LIN {X 0,Y 573.931,Z 295.333,A -85,B 0,C 180,E1 -2262.553,E2 -2262.553} C_VEL
LIN {X 0,Y 573.875,Z 198.299,A -85,B 0,C 180,E1 -2263.776,E2 -2263.776} C_VEL
LIN {X 0,Y 573.396,Z 194.795,A -85,B 0,C 180,E1 -2263.85,E2 -2263.85} C_VEL
LIN {X 0,Y 573.536,Z 174.901,A -85,B 0,C 180,E1 -2266.722,E2 -2266.722} C_VEL
LIN {X 0,Y 573.71,Z 157.017,A -85,B 0,C 180,E1 -2269.314,E2 -2269.314} C_VEL
LIN {X 0,Y 573.882,Z 139.078,A -85,B 0,C 180,E1 -2271.932,E2 -2271.932} C_VEL
LIN {X 0,Y 573.502,Z 133.913,A -85,B 0,C 180,E1 -2272.706,E2 -2272.706} C_VEL
LIN {X 0,Y 573.198,Z 132.088,A -85,B 0,C 180,E1 -2273.017,E2 -2273.017} C_VEL
LIN {X 0,Y 573.2,Z 132.089,A -85,B 0,C 180,E1 -2275.412,E2 -2275.412} C_VEL
LIN {X 0,Y 573.191,Z 132.083,A -85,B 0,C 180,E1 -2278.017,E2 -2278.017} C_VEL
LIN {X 0,Y 573.199,Z 132.085,A -85,B 0,C 180,E1 -2280.877,E2 -2280.877} C_VEL
LIN {X 0,Y 573.24,Z 132.08,A -85,B 0,C 180,E1 -2283.52,E2 -2283.52} C_VEL
LIN {X 0,Y 573.175,Z 132.083,A -85,B 0,C 180,E1 -2286.054,E2 -2286.054} C_VEL
LIN {X 0,Y 573.223,Z 132.081,A -85,B 0,C 180,E1 -2288.702,E2 -2288.702} C_VEL
LIN {X 0,Y 573.19,Z 132.083,A -85,B 0,C 180,E1 -2291.588,E2 -2291.588} C_VEL
LIN {X 0,Y 573.203,Z 132.085,A -85,B 0,C 180,E1 -2294.672,E2 -2294.672} C_VEL
LIN {X 0,Y 573.2,Z 132.08,A -85,B 0,C 180,E1 -2297.596,E2 -2297.596} C_VEL
LIN {X 0,Y 573.225,Z 132.082,A -85,B 0,C 180,E1 -2300.569,E2 -2300.569} C_VEL
LIN {X 0,Y 573.221,Z 132.081,A -85,B 0,C 180,E1 -2303.075,E2 -2303.075} C_VEL
LIN {X 0,Y 573.235,Z 132.075,A -85,B 0,C 180,E1 -2305.669,E2 -2305.669} C_VEL
LIN {X 0,Y 573.212,Z 132.08,A -85,B 0,C 180,E1 -2308.182,E2 -2308.182} C_VEL
LIN {X 0,Y 573.207,Z 132.087,A -85,B 0,C 180,E1 -2310.631,E2 -2310.631} C_VEL
LIN {X 0,Y 573.194,Z 132.079,A -85,B 0,C 180,E1 -2313.514,E2 -2313.514} C_VEL
LIN {X 0,Y 573.184,Z 132.086,A -85,B 0,C 180,E1 -2316.132,E2 -2316.132} C_VEL
LIN {X 0,Y 573.21,Z 132.079,A -85,B 0,C 180,E1 -2319.172,E2 -2319.172} C_VEL
LIN {X 0,Y 573.182,Z 132.081,A -85,B 0,C 180,E1 -2321.41,E2 -2321.41} C_VEL
LIN {X 0,Y 573.194,Z 132.088,A -85,B 0,C 180,E1 -2324.351,E2 -2324.351} C_VEL
LIN {X 0,Y 573.184,Z 132.087,A -85,B 0,C 180,E1 -2326.528,E2 -2326.528} C_VEL
LIN {X 0,Y 573.233,Z 132.075,A -85,B 0,C 180,E1 -2329.402,E2 -2329.402} C_VEL
LIN {X 0,Y 573.21,Z 132.086,A -85,B 0,C 180,E1 -2332.249,E2 -2332.249} C_VEL
LIN {X 0,Y 573.264,Z 132.07,A -85,B 0,C 180,E1 -2335.077,E2 -2335.077} C_VEL
LIN {X 0,Y 573.303,Z 132.075,A -85,B 0,C 180,E1 -2337.892,E2 -2337.892} C_VEL
LIN {X 0,Y 573.309,Z 132.075,A -85,B 0,C 180,E1 -2340,E2 -2340} C_VEL
LIN {X 0,Y 573.261,Z 132.072,A -85,B 0,C 180,E1 -2342.811,E2 -2342.811} C_VEL
LIN {X 0,Y 573.261,Z 132.079,A -85,B 0,C 180,E1 -2345.628,E2 -2345.628} C_VEL
LIN {X 0,Y 573.225,Z 132.078,A -85,B 0,C 180,E1 -2348.46,E2 -2348.46} C_VEL
LIN {X 0,Y 573.226,Z 132.081,A -85,B 0,C 180,E1 -2351.313,E2 -2351.313} C_VEL
LIN {X 0,Y 573.247,Z 132.075,A -85,B 0,C 180,E1 -2354.414,E2 -2354.414} C_VEL
LIN {X 0,Y 573.165,Z 132.088,A -85,B 0,C 180,E1 -2357.114,E2 -2357.114} C_VEL
LIN {X 0,Y 573.255,Z 132.08,A -85,B 0,C 180,E1 -2359.33,E2 -2359.33} C_VEL
LIN {X 0,Y 573.187,Z 132.083,A -85,B 0,C 180,E1 -2362.339,E2 -2362.339} C_VEL
LIN {X 0,Y 573.192,Z 132.086,A -85,B 0,C 180,E1 -2363.279,E2 -2363.279} C_VEL
LIN {X 0,Y 572.863,Z 132.396,A -85,B 0,C 180,E1 -2363.667,E2 -2363.667} C_VEL
LIN {X 0,Y 571.545,Z 133.798,A -85,B 0,C 180,E1 -2364.226,E2 -2364.226} C_VEL
LIN {X 0,Y 569.755,Z 135.989,A -85,B 0,C 180,E1 -2364.752,E2 -2364.752} C_VEL
LIN {X 0,Y 567.024,Z 140.741,A -85,B 0,C 180,E1 -2365.613,E2 -2365.613} C_VEL
LIN {X 0,Y 566.439,Z 143.796,A -85,B 0,C 180,E1 -2366.138,E2 -2366.138} C_VEL
LIN {X 0,Y 566.337,Z 160.929,A -85,B 0,C 180,E1 -2369.129,E2 -2369.129} C_VEL
LIN {X 0,Y 566.28,Z 166.18,A -85,B 0,C 180,E1 -2370.051,E2 -2370.051} C_VEL
LIN {X 0,Y 567.205,Z 173.364,A -85,B 0,C 180,E1 -2370.168,E2 -2370.168} C_VEL
LIN {X 0,Y 566.947,Z 273.932,A -85,B 0,C 180,E1 -2371.466,E2 -2371.466} C_VEL
LIN {X 0,Y 566.823,Z 285.922,A -85,B 0,C 180,E1 -2371.76,E2 -2371.76} C_VEL
LIN {X 0,Y 566.764,Z 296.329,A -85,B 0,C 180,E1 -2372.117,E2 -2372.117} C_VEL
LIN {X 0,Y 566.623,Z 306.781,A -85,B 0,C 180,E1 -2372.583,E2 -2372.583} C_VEL
LIN {X 0,Y 566.446,Z 317.622,A -85,B 0,C 180,E1 -2373.193,E2 -2373.193} C_VEL
LIN {X 0,Y 566.316,Z 329.517,A -85,B 0,C 180,E1 -2374.056,E2 -2374.056} C_VEL
LIN {X 0,Y 566.245,Z 338.018,A -85,B 0,C 180,E1 -2374.815,E2 -2374.815} C_VEL
LIN {X 0,Y 566.139,Z 344.619,A -85,B 0,C 180,E1 -2375.504,E2 -2375.504} C_VEL
LIN {X 0,Y 566.063,Z 351.559,A -85,B 0,C 180,E1 -2376.362,E2 -2376.362} C_VEL
LIN {X 0,Y 565.983,Z 358.32,A -85,B 0,C 180,E1 -2377.374,E2 -2377.374} C_VEL
LIN {X 0,Y 565.975,Z 363.801,A -85,B 0,C 180,E1 -2378.38,E2 -2378.38} C_VEL
LIN {X 0,Y 565.888,Z 367.871,A -85,B 0,C 180,E1 -2379.3,E2 -2379.3} C_VEL
LIN {X 0,Y 565.901,Z 372.701,A -85,B 0,C 180,E1 -2380.751,E2 -2380.751} C_VEL
LIN {X 0,Y 565.861,Z 375.529,A -85,B 0,C 180,E1 -2382.119,E2 -2382.119} C_VEL
LIN {X 0,Y 565.845,Z 376.629,A -85,B 0,C 180,E1 -2383.087,E2 -2383.087} C_VEL
LIN {X 0,Y 565.858,Z 376.999,A -85,B 0,C 180,E1 -2384.069,E2 -2384.069} C_VEL
LIN {X 0,Y 565.875,Z 376.587,A -85,B 0,C 180,E1 -2385.066,E2 -2385.066} C_VEL
LIN {X 0,Y 565.852,Z 375.359,A -85,B 0,C 180,E1 -2386.085,E2 -2386.085} C_VEL
LIN {X 0,Y 565.901,Z 372.206,A -85,B 0,C 180,E1 -2387.505,E2 -2387.505} C_VEL
LIN {X 0,Y 565.921,Z 368.981,A -85,B 0,C 180,E1 -2388.505,E2 -2388.505} C_VEL
LIN {X 0,Y 565.944,Z 364.768,A -85,B 0,C 180,E1 -2389.512,E2 -2389.512} C_VEL
LIN {X 0,Y 566.014,Z 359.438,A -85,B 0,C 180,E1 -2390.528,E2 -2390.528} C_VEL
LIN {X 0,Y 566.022,Z 353.429,A -85,B 0,C 180,E1 -2391.465,E2 -2391.465} C_VEL
LIN {X 0,Y 566.111,Z 346.956,A -85,B 0,C 180,E1 -2392.309,E2 -2392.309} C_VEL
LIN {X 0,Y 566.208,Z 339.781,A -85,B 0,C 180,E1 -2393.099,E2 -2393.099} C_VEL
LIN {X 0,Y 566.346,Z 332.677,A -85,B 0,C 180,E1 -2393.765,E2 -2393.765} C_VEL
LIN {X 0,Y 566.39,Z 324.604,A -85,B 0,C 180,E1 -2394.413,E2 -2394.413} C_VEL
LIN {X 0,Y 566.516,Z 315.348,A -85,B 0,C 180,E1 -2395.031,E2 -2395.031} C_VEL
LIN {X 0,Y 566.609,Z 306.216,A -85,B 0,C 180,E1 -2395.535,E2 -2395.535} C_VEL
LIN {X 0,Y 566.726,Z 296.359,A -85,B 0,C 180,E1 -2395.973,E2 -2395.973} C_VEL
LIN {X 0,Y 566.82,Z 285.576,A -85,B 0,C 180,E1 -2396.34,E2 -2396.34} C_VEL
LIN {X 0,Y 566.935,Z 273.792,A -85,B 0,C 180,E1 -2396.627,E2 -2396.627} C_VEL
LIN {X 0,Y 567.061,Z 171.116,A -85,B 0,C 180,E1 -2397.954,E2 -2397.954} C_VEL
LIN {X 0,Y 566.232,Z 166.076,A -85,B 0,C 180,E1 -2398.059,E2 -2398.059} C_VEL
LIN {X 0,Y 566.436,Z 150.118,A -85,B 0,C 180,E1 -2400.87,E2 -2400.87} C_VEL
LIN {X 0,Y 566.555,Z 135.482,A -85,B 0,C 180,E1 -2403.477,E2 -2403.477} C_VEL
LIN {X 0,Y 566.18,Z 132.961,A -85,B 0,C 180,E1 -2403.953,E2 -2403.953} C_VEL
LIN {X 0,Y 566.142,Z 132.968,A -85,B 0,C 180,E1 -2406.725,E2 -2406.725} C_VEL
LIN {X 0,Y 566.184,Z 132.958,A -85,B 0,C 180,E1 -2408.902,E2 -2408.902} C_VEL
LIN {X 0,Y 566.177,Z 132.955,A -85,B 0,C 180,E1 -2411.172,E2 -2411.172} C_VEL
LIN {X 0,Y 566.164,Z 132.961,A -85,B 0,C 180,E1 -2414.152,E2 -2414.152} C_VEL
LIN {X 0,Y 566.156,Z 132.966,A -85,B 0,C 180,E1 -2416.358,E2 -2416.358} C_VEL
LIN {X 0,Y 566.206,Z 132.95,A -85,B 0,C 180,E1 -2419.27,E2 -2419.27} C_VEL
LIN {X 0,Y 566.183,Z 132.961,A -85,B 0,C 180,E1 -2422.152,E2 -2422.152} C_VEL
LIN {X 0,Y 566.245,Z 132.946,A -85,B 0,C 180,E1 -2425.016,E2 -2425.016} C_VEL
LIN {X 0,Y 566.275,Z 132.947,A -85,B 0,C 180,E1 -2427.866,E2 -2427.866} C_VEL
LIN {X 0,Y 566.282,Z 132.949,A -85,B 0,C 180,E1 -2430,E2 -2430} C_VEL
LIN {X 0,Y 566.234,Z 132.947,A -85,B 0,C 180,E1 -2432.846,E2 -2432.846} C_VEL
LIN {X 0,Y 566.232,Z 132.953,A -85,B 0,C 180,E1 -2435.699,E2 -2435.699} C_VEL
LIN {X 0,Y 566.182,Z 132.954,A -85,B 0,C 180,E1 -2438.566,E2 -2438.566} C_VEL
LIN {X 0,Y 566.189,Z 132.956,A -85,B 0,C 180,E1 -2441.455,E2 -2441.455} C_VEL
LIN {X 0,Y 566.199,Z 132.952,A -85,B 0,C 180,E1 -2444.494,E2 -2444.494} C_VEL
LIN {X 0,Y 566.153,Z 132.961,A -85,B 0,C 180,E1 -2447.333,E2 -2447.333} C_VEL
LIN {X 0,Y 566.17,Z 132.964,A -85,B 0,C 180,E1 -2449.582,E2 -2449.582} C_VEL
LIN {X 0,Y 566.141,Z 132.964,A -85,B 0,C 180,E1 -2451.864,E2 -2451.864} C_VEL
LIN {X 0,Y 566.174,Z 132.957,A -85,B 0,C 180,E1 -2455.021,E2 -2455.021} C_VEL
LIN {X 0,Y 566.154,Z 132.965,A -85,B 0,C 180,E1 -2457.342,E2 -2457.342} C_VEL
LIN {X 0,Y 566.142,Z 132.963,A -85,B 0,C 180,E1 -2459.772,E2 -2459.772} C_VEL
LIN {X 0,Y 566.185,Z 132.953,A -85,B 0,C 180,E1 -2462.427,E2 -2462.427} C_VEL
LIN {X 0,Y 566.156,Z 132.961,A -85,B 0,C 180,E1 -2464.986,E2 -2464.986} C_VEL
LIN {X 0,Y 566.182,Z 132.96,A -85,B 0,C 180,E1 -2467.461,E2 -2467.461} C_VEL
LIN {X 0,Y 566.188,Z 132.953,A -85,B 0,C 180,E1 -2470.2,E2 -2470.2} C_VEL
LIN {X 0,Y 566.17,Z 132.964,A -85,B 0,C 180,E1 -2473.056,E2 -2473.056} C_VEL
LIN {X 0,Y 566.148,Z 132.957,A -85,B 0,C 180,E1 -2476.053,E2 -2476.053} C_VEL
LIN {X 0,Y 566.148,Z 132.965,A -85,B 0,C 180,E1 -2478.858,E2 -2478.858} C_VEL
LIN {X 0,Y 566.191,Z 132.955,A -85,B 0,C 180,E1 -2481.444,E2 -2481.444} C_VEL
LIN {X 0,Y 566.128,Z 132.962,A -85,B 0,C 180,E1 -2484.306,E2 -2484.306} C_VEL
LIN {X 0,Y 566.184,Z 132.962,A -85,B 0,C 180,E1 -2486.896,E2 -2486.896} C_VEL
LIN {X 0,Y 566.15,Z 132.959,A -85,B 0,C 180,E1 -2489.406,E2 -2489.406} C_VEL
LIN {X 0,Y 566.133,Z 132.96,A -85,B 0,C 180,E1 -2491.854,E2 -2491.854} C_VEL
LIN {X 0,Y 566.179,Z 132.957,A -85,B 0,C 180,E1 -2494.25,E2 -2494.25} C_VEL
LIN {X 0,Y 566.13,Z 132.96,A -85,B 0,C 180,E1 -2497.367,E2 -2497.367} C_VEL
LIN {X 0,Y 566.16,Z 132.956,A -85,B 0,C 180,E1 -2499.661,E2 -2499.661} C_VEL
LIN {X 0,Y 566.153,Z 132.959,A -85,B 0,C 180,E1 -2501.921,E2 -2501.921} C_VEL
LIN {X 0,Y 566.171,Z 132.957,A -85,B 0,C 180,E1 -2504.89,E2 -2504.89} C_VEL
LIN {X 0,Y 566.164,Z 132.958,A -85,B 0,C 180,E1 -2507.818,E2 -2507.818} C_VEL
LIN {X 0,Y 566.152,Z 132.962,A -85,B 0,C 180,E1 -2509.992,E2 -2509.992} C_VEL
LIN {X 0,Y 566.175,Z 132.955,A -85,B 0,C 180,E1 -2512.87,E2 -2512.87} C_VEL
LIN {X 0,Y 566.242,Z 132.946,A -85,B 0,C 180,E1 -2515.016,E2 -2515.016} C_VEL
LIN {X 0,Y 566.273,Z 132.948,A -85,B 0,C 180,E1 -2517.867,E2 -2517.867} C_VEL
LIN {X 0,Y 566.279,Z 132.95,A -85,B 0,C 180,E1 -2520,E2 -2520} C_VEL
LIN {X 0,Y 566.231,Z 132.947,A -85,B 0,C 180,E1 -2522.846,E2 -2522.846} C_VEL
LIN {X 0,Y 566.23,Z 132.953,A -85,B 0,C 180,E1 -2525.699,E2 -2525.699} C_VEL
LIN {X 0,Y 566.179,Z 132.955,A -85,B 0,C 180,E1 -2528.567,E2 -2528.567} C_VEL
LIN {X 0,Y 566.186,Z 132.957,A -85,B 0,C 180,E1 -2531.456,E2 -2531.456} C_VEL
LIN {X 0,Y 566.197,Z 132.952,A -85,B 0,C 180,E1 -2534.494,E2 -2534.494} C_VEL
LIN {X 0,Y 566.151,Z 132.962,A -85,B 0,C 180,E1 -2537.333,E2 -2537.333} C_VEL
LIN {X 0,Y 566.168,Z 132.965,A -85,B 0,C 180,E1 -2539.582,E2 -2539.582} C_VEL
LIN {X 0,Y 566.14,Z 132.964,A -85,B 0,C 180,E1 -2541.865,E2 -2541.865} C_VEL
LIN {X 0,Y 566.173,Z 132.957,A -85,B 0,C 180,E1 -2545.022,E2 -2545.022} C_VEL
LIN {X 0,Y 566.153,Z 132.965,A -85,B 0,C 180,E1 -2547.342,E2 -2547.342} C_VEL
LIN {X 0,Y 566.141,Z 132.962,A -85,B 0,C 180,E1 -2549.773,E2 -2549.773} C_VEL
LIN {X 0,Y 566.185,Z 132.953,A -85,B 0,C 180,E1 -2552.428,E2 -2552.428} C_VEL
LIN {X 0,Y 566.154,Z 132.962,A -85,B 0,C 180,E1 -2554.987,E2 -2554.987} C_VEL
LIN {X 0,Y 566.184,Z 132.959,A -85,B 0,C 180,E1 -2557.462,E2 -2557.462} C_VEL
LIN {X 0,Y 566.162,Z 132.956,A -85,B 0,C 180,E1 -2560.203,E2 -2560.203} C_VEL
LIN {X 0,Y 566.144,Z 132.968,A -85,B 0,C 180,E1 -2563.06,E2 -2563.06} C_VEL
LIN {X 0,Y 566.151,Z 132.957,A -85,B 0,C 180,E1 -2566.054,E2 -2566.054} C_VEL
LIN {X 0,Y 566.141,Z 132.967,A -85,B 0,C 180,E1 -2568.858,E2 -2568.858} C_VEL
LIN {X 0,Y 566.168,Z 132.956,A -85,B 0,C 180,E1 -2571.636,E2 -2571.636} C_VEL
LIN {X 0,Y 566.129,Z 132.962,A -85,B 0,C 180,E1 -2574.306,E2 -2574.306} C_VEL
LIN {X 0,Y 566.16,Z 132.965,A -85,B 0,C 180,E1 -2576.894,E2 -2576.894} C_VEL
LIN {X 0,Y 566.147,Z 132.959,A -85,B 0,C 180,E1 -2579.406,E2 -2579.406} C_VEL
LIN {X 0,Y 566.139,Z 132.96,A -85,B 0,C 180,E1 -2581.854,E2 -2581.854} C_VEL
LIN {X 0,Y 566.171,Z 132.959,A -85,B 0,C 180,E1 -2584.249,E2 -2584.249} C_VEL
LIN {X 0,Y 566.158,Z 133.045,A -85,B 0,C 180,E1 -2586.833,E2 -2586.833} C_VEL
LIN {X 0,Y 566.938,Z 137.862,A -85,B 0,C 180,E1 -2587.593,E2 -2587.593} C_VEL
LIN {X 0,Y 566.777,Z 155.67,A -85,B 0,C 180,E1 -2590.251,E2 -2590.251} C_VEL
LIN {X 0,Y 566.546,Z 172.886,A -85,B 0,C 180,E1 -2592.783,E2 -2592.783} C_VEL
LIN {X 0,Y 566.406,Z 192.432,A -85,B 0,C 180,E1 -2595.631,E2 -2595.631} C_VEL
LIN {X 0,Y 566.422,Z 195.149,A -85,B 0,C 180,E1 -2595.998,E2 -2595.998} C_VEL
LIN {X 0,Y 567.176,Z 200.341,A -85,B 0,C 180,E1 -2596.084,E2 -2596.084} C_VEL
LIN {X 0,Y 566.98,Z 302.95,A -85,B 0,C 180,E1 -2597.404,E2 -2597.404} C_VEL
LIN {X 0,Y 566.841,Z 316.219,A -85,B 0,C 180,E1 -2597.719,E2 -2597.719} C_VEL
LIN {X 0,Y 566.743,Z 328.379,A -85,B 0,C 180,E1 -2598.148,E2 -2598.148} C_VEL
LIN {X 0,Y 566.603,Z 340.366,A -85,B 0,C 180,E1 -2598.72,E2 -2598.72} C_VEL
LIN {X 0,Y 566.439,Z 352.196,A -85,B 0,C 180,E1 -2599.455,E2 -2599.455} C_VEL
LIN {X 0,Y 566.325,Z 362.605,A -85,B 0,C 180,E1 -2600.265,E2 -2600.265} C_VEL
LIN {X 0,Y 566.207,Z 371.113,A -85,B 0,C 180,E1 -2601.074,E2 -2601.074} C_VEL
LIN {X 0,Y 566.112,Z 378.961,A -85,B 0,C 180,E1 -2601.972,E2 -2601.972} C_VEL
LIN {X 0,Y 566.004,Z 386.623,A -85,B 0,C 180,E1 -2603.047,E2 -2603.047} C_VEL
LIN {X 0,Y 566.004,Z 393.679,A -85,B 0,C 180,E1 -2604.299,E2 -2604.299} C_VEL
LIN {X 0,Y 565.933,Z 398.372,A -85,B 0,C 180,E1 -2605.37,E2 -2605.37} C_VEL
LIN {X 0,Y 565.927,Z 401.958,A -85,B 0,C 180,E1 -2606.44,E2 -2606.44} C_VEL
LIN {X 0,Y 565.878,Z 403.807,A -85,B 0,C 180,E1 -2607.152,E2 -2607.152} C_VEL
LIN {X 0,Y 565.846,Z 406.184,A -85,B 0,C 180,E1 -2608.576,E2 -2608.576} C_VEL
LIN {X 0,Y 565.839,Z 407,A -85,B 0,C 180,E1 -2610,E2 -2610} C_VEL
LIN {X 0,Y 565.846,Z 406.185,A -85,B 0,C 180,E1 -2611.423,E2 -2611.423} C_VEL
LIN {X 0,Y 565.878,Z 403.81,A -85,B 0,C 180,E1 -2612.847,E2 -2612.847} C_VEL
LIN {X 0,Y 565.926,Z 400.896,A -85,B 0,C 180,E1 -2613.916,E2 -2613.916} C_VEL
LIN {X 0,Y 565.878,Z 396.949,A -85,B 0,C 180,E1 -2614.987,E2 -2614.987} C_VEL
LIN {X 0,Y 566.002,Z 391.868,A -85,B 0,C 180,E1 -2616.058,E2 -2616.058} C_VEL
LIN {X 0,Y 566.04,Z 385.469,A -85,B 0,C 180,E1 -2617.132,E2 -2617.132} C_VEL
LIN {X 0,Y 566.134,Z 377.479,A -85,B 0,C 180,E1 -2618.207,E2 -2618.207} C_VEL
LIN {X 0,Y 566.229,Z 369.336,A -85,B 0,C 180,E1 -2619.105,E2 -2619.105} C_VEL
LIN {X 0,Y 566.347,Z 359.402,A -85,B 0,C 180,E1 -2620.005,E2 -2620.005} C_VEL
LIN {X 0,Y 566.536,Z 348.295,A -85,B 0,C 180,E1 -2620.807,E2 -2620.807} C_VEL
LIN {X 0,Y 566.612,Z 337.178,A -85,B 0,C 180,E1 -2621.446,E2 -2621.446} C_VEL
LIN {X 0,Y 566.745,Z 324.986,A -85,B 0,C 180,E1 -2621.988,E2 -2621.988} C_VEL
LIN {X 0,Y 566.917,Z 312.186,A -85,B 0,C 180,E1 -2622.393,E2 -2622.393} C_VEL
LIN {X 0,Y 566.994,Z 300.124,A -85,B 0,C 180,E1 -2622.641,E2 -2622.641} C_VEL
LIN {X 0,Y 567.04,Z 199.447,A -85,B 0,C 180,E1 -2623.931,E2 -2623.931} C_VEL
LIN {X 0,Y 566.391,Z 194.795,A -85,B 0,C 180,E1 -2624.025,E2 -2624.025} C_VEL
LIN {X 0,Y 566.55,Z 175.031,A -85,B 0,C 180,E1 -2626.895,E2 -2626.895} C_VEL
LIN {X 0,Y 566.73,Z 156.765,A -85,B 0,C 180,E1 -2629.562,E2 -2629.562} C_VEL
LIN {X 0,Y 566.912,Z 138.815,A -85,B 0,C 180,E1 -2632.216,E2 -2632.216} C_VEL
LIN {X 0,Y 566.155,Z 132.966,A -85,B 0,C 180,E1 -2633.142,E2 -2633.142} C_VEL
LIN {X 0,Y 566.17,Z 132.961,A -85,B 0,C 180,E1 -2635.751,E2 -2635.751} C_VEL
LIN {X 0,Y 566.136,Z 132.961,A -85,B 0,C 180,E1 -2638.189,E2 -2638.189} C_VEL
LIN {X 0,Y 566.167,Z 132.964,A -85,B 0,C 180,E1 -2641.072,E2 -2641.072} C_VEL
LIN {X 0,Y 566.193,Z 132.955,A -85,B 0,C 180,E1 -2643.731,E2 -2643.731} C_VEL
LIN {X 0,Y 566.142,Z 132.961,A -85,B 0,C 180,E1 -2646.573,E2 -2646.573} C_VEL
LIN {X 0,Y 566.199,Z 132.959,A -85,B 0,C 180,E1 -2649.274,E2 -2649.274} C_VEL
LIN {X 0,Y 566.139,Z 132.96,A -85,B 0,C 180,E1 -2652.093,E2 -2652.093} C_VEL
LIN {X 0,Y 566.16,Z 132.965,A -85,B 0,C 180,E1 -2655.036,E2 -2655.036} C_VEL
LIN {X 0,Y 566.136,Z 132.96,A -85,B 0,C 180,E1 -2658.144,E2 -2658.144} C_VEL
LIN {X 0,Y 566.197,Z 132.96,A -85,B 0,C 180,E1 -2660.725,E2 -2660.725} C_VEL
LIN {X 0,Y 566.142,Z 132.959,A -85,B 0,C 180,E1 -2663.425,E2 -2663.425} C_VEL
LIN {X 0,Y 566.189,Z 132.956,A -85,B 0,C 180,E1 -2666.268,E2 -2666.268} C_VEL
LIN {X 0,Y 566.165,Z 132.96,A -85,B 0,C 180,E1 -2668.926,E2 -2668.926} C_VEL
LIN {X 0,Y 566.133,Z 132.96,A -85,B 0,C 180,E1 -2671.853,E2 -2671.853} C_VEL
LIN {X 0,Y 566.18,Z 132.958,A -85,B 0,C 180,E1 -2674.249,E2 -2674.249} C_VEL
LIN {X 0,Y 566.14,Z 132.963,A -85,B 0,C 180,E1 -2676.724,E2 -2676.724} C_VEL
LIN {X 0,Y 566.175,Z 132.957,A -85,B 0,C 180,E1 -2678.901,E2 -2678.901} C_VEL
LIN {X 0,Y 566.159,Z 132.956,A -85,B 0,C 180,E1 -2681.17,E2 -2681.17} C_VEL
LIN {X 0,Y 566.161,Z 132.964,A -85,B 0,C 180,E1 -2684.151,E2 -2684.151} C_VEL
LIN {X 0,Y 566.152,Z 132.966,A -85,B 0,C 180,E1 -2686.357,E2 -2686.357} C_VEL
LIN {X 0,Y 566.203,Z 132.951,A -85,B 0,C 180,E1 -2689.269,E2 -2689.269} C_VEL
LIN {X 0,Y 566.178,Z 132.963,A -85,B 0,C 180,E1 -2692.152,E2 -2692.152} C_VEL
LIN {X 0,Y 566.24,Z 132.945,A -85,B 0,C 180,E1 -2695.015,E2 -2695.015} C_VEL
LIN {X 0,Y 566.272,Z 132.95,A -85,B 0,C 180,E1 -2697.866,E2 -2697.866} C_VEL
LIN {X 0,Y 566.277,Z 132.95,A -85,B 0,C 180,E1 -2700,E2 -2700} C_VEL
LIN {X 0,Y 566.229,Z 132.948,A -85,B 0,C 180,E1 -2702.845,E2 -2702.845} C_VEL
LIN {X 0,Y 566.23,Z 132.956,A -85,B 0,C 180,E1 -2705.698,E2 -2705.698} C_VEL
LIN {X 0,Y 566.177,Z 132.955,A -85,B 0,C 180,E1 -2708.566,E2 -2708.566} C_VEL
LIN {X 0,Y 566.183,Z 132.961,A -85,B 0,C 180,E1 -2711.455,E2 -2711.455} C_VEL
LIN {X 0,Y 566.203,Z 132.953,A -85,B 0,C 180,E1 -2714.497,E2 -2714.497} C_VEL
LIN {X 0,Y 566.139,Z 132.966,A -85,B 0,C 180,E1 -2717.333,E2 -2717.333} C_VEL
LIN {X 0,Y 566.187,Z 132.963,A -85,B 0,C 180,E1 -2719.581,E2 -2719.581} C_VEL
LIN {X 0,Y 566.14,Z 132.965,A -85,B 0,C 180,E1 -2721.864,E2 -2721.864} C_VEL
LIN {X 0,Y 566.179,Z 133.046,A -85,B 0,C 180,E1 -2724.279,E2 -2724.279} C_VEL
LIN {X 0,Y 566.495,Z 137.739,A -85,B 0,C 180,E1 -2725.092,E2 -2725.092} C_VEL
LIN {X 0,Y 566.439,Z 143.796,A -85,B 0,C 180,E1 -2726.138,E2 -2726.138} C_VEL
LIN {X 0,Y 565.819,Z 146.819,A -85,B 0,C 180,E1 -2726.647,E2 -2726.647} C_VEL
LIN {X 0,Y 562.955,Z 151.99,A -85,B 0,C 180,E1 -2727.456,E2 -2727.456} C_VEL
LIN {X 0,Y 560.027,Z 157.182,A -85,B 0,C 180,E1 -2728.272,E2 -2728.272} C_VEL
LIN {X 0,Y 559.328,Z 160.192,A -85,B 0,C 180,E1 -2728.789,E2 -2728.789} C_VEL
LIN {X 0,Y 559.233,Z 166.292,A -85,B 0,C 180,E1 -2729.874,E2 -2729.874} C_VEL
LIN {X 0,Y 560.329,Z 174.113,A -85,B 0,C 180,E1 -2730.004,E2 -2730.004} C_VEL
LIN {X 0,Y 560.055,Z 273.245,A -85,B 0,C 180,E1 -2731.296,E2 -2731.296} C_VEL
LIN {X 0,Y 559.909,Z 284.947,A -85,B 0,C 180,E1 -2731.578,E2 -2731.578} C_VEL
LIN {X 0,Y 559.807,Z 295.31,A -85,B 0,C 180,E1 -2731.927,E2 -2731.927} C_VEL
LIN {X 0,Y 559.67,Z 305.191,A -85,B 0,C 180,E1 -2732.361,E2 -2732.361} C_VEL
LIN {X 0,Y 559.524,Z 314.402,A -85,B 0,C 180,E1 -2732.864,E2 -2732.864} C_VEL
LIN {X 0,Y 559.4,Z 323.117,A -85,B 0,C 180,E1 -2733.44,E2 -2733.44} C_VEL
LIN {X 0,Y 559.308,Z 330.635,A -85,B 0,C 180,E1 -2734.026,E2 -2734.026} C_VEL
LIN {X 0,Y 559.195,Z 338.709,A -85,B 0,C 180,E1 -2734.769,E2 -2734.769} C_VEL
LIN {X 0,Y 559.095,Z 345.863,A -85,B 0,C 180,E1 -2735.547,E2 -2735.547} C_VEL
LIN {X 0,Y 558.995,Z 352.677,A -85,B 0,C 180,E1 -2736.426,E2 -2736.426} C_VEL
LIN {X 0,Y 558.911,Z 358.761,A -85,B 0,C 180,E1 -2737.366,E2 -2737.366} C_VEL
LIN {X 0,Y 558.892,Z 364.246,A -85,B 0,C 180,E1 -2738.403,E2 -2738.403} C_VEL
LIN {X 0,Y 558.802,Z 368.591,A -85,B 0,C 180,E1 -2739.429,E2 -2739.429} C_VEL
LIN {X 0,Y 558.806,Z 371.692,A -85,B 0,C 180,E1 -2740.368,E2 -2740.368} C_VEL
LIN {X 0,Y 558.788,Z 373.433,A -85,B 0,C 180,E1 -2741.008,E2 -2741.008} C_VEL
LIN {X 0,Y 558.761,Z 375.515,A -85,B 0,C 180,E1 -2742.091,E2 -2742.091} C_VEL
LIN {X 0,Y 558.759,Z 376.672,A -85,B 0,C 180,E1 -2743.155,E2 -2743.155} C_VEL
LIN {X 0,Y 558.774,Z 376.972,A -85,B 0,C 180,E1 -2744.2,E2 -2744.2} C_VEL
LIN {X 0,Y 558.784,Z 376.456,A -85,B 0,C 180,E1 -2745.226,E2 -2745.226} C_VEL
LIN {X 0,Y 558.76,Z 375.174,A -85,B 0,C 180,E1 -2746.23,E2 -2746.23} C_VEL
LIN {X 0,Y 558.773,Z 373.114,A -85,B 0,C 180,E1 -2747.221,E2 -2747.221} C_VEL
LIN {X 0,Y 558.823,Z 370.284,A -85,B 0,C 180,E1 -2748.2,E2 -2748.2} C_VEL
LIN {X 0,Y 558.862,Z 365.631,A -85,B 0,C 180,E1 -2749.4,E2 -2749.4} C_VEL
LIN {X 0,Y 558.939,Z 359.588,A -85,B 0,C 180,E1 -2750.583,E2 -2750.583} C_VEL
LIN {X 0,Y 558.971,Z 354.502,A -85,B 0,C 180,E1 -2751.405,E2 -2751.405} C_VEL
LIN {X 0,Y 559.044,Z 347.29,A -85,B 0,C 180,E1 -2752.372,E2 -2752.372} C_VEL
LIN {X 0,Y 559.161,Z 341.184,A -85,B 0,C 180,E1 -2753.07,E2 -2753.07} C_VEL
LIN {X 0,Y 559.305,Z 332.375,A -85,B 0,C 180,E1 -2753.914,E2 -2753.914} C_VEL
LIN {X 0,Y 559.395,Z 324.008,A -85,B 0,C 180,E1 -2754.586,E2 -2754.586} C_VEL
LIN {X 0,Y 559.516,Z 315.753,A -85,B 0,C 180,E1 -2755.145,E2 -2755.145} C_VEL
LIN {X 0,Y 559.638,Z 306.899,A -85,B 0,C 180,E1 -2755.645,E2 -2755.645} C_VEL
LIN {X 0,Y 559.768,Z 296.43,A -85,B 0,C 180,E1 -2756.12,E2 -2756.12} C_VEL
LIN {X 0,Y 559.884,Z 286.241,A -85,B 0,C 180,E1 -2756.475,E2 -2756.475} C_VEL
LIN {X 0,Y 560.016,Z 274.242,A -85,B 0,C 180,E1 -2756.776,E2 -2756.776} C_VEL
LIN {X 0,Y 560.169,Z 217.742,A -85,B 0,C 180,E1 -2757.525,E2 -2757.525} C_VEL
LIN {X 0,Y 560.172,Z 171.726,A -85,B 0,C 180,E1 -2758.123,E2 -2758.123} C_VEL
LIN {X 0,Y 559.232,Z 166.277,A -85,B 0,C 180,E1 -2758.221,E2 -2758.221} C_VEL
LIN {X 0,Y 559.426,Z 150.276,A -85,B 0,C 180,E1 -2761.075,E2 -2761.075} C_VEL
LIN {X 0,Y 559.571,Z 136.646,A -85,B 0,C 180,E1 -2763.522,E2 -2763.522} C_VEL
LIN {X 0,Y 559.147,Z 133.838,A -85,B 0,C 180,E1 -2764.052,E2 -2764.052} C_VEL
LIN {X 0,Y 559.086,Z 133.842,A -85,B 0,C 180,E1 -2767.066,E2 -2767.066} C_VEL
LIN {X 0,Y 559.142,Z 133.831,A -85,B 0,C 180,E1 -2769.394,E2 -2769.394} C_VEL
LIN {X 0,Y 559.108,Z 133.835,A -85,B 0,C 180,E1 -2771.685,E2 -2771.685} C_VEL
LIN {X 0,Y 559.123,Z 133.838,A -85,B 0,C 180,E1 -2774.695,E2 -2774.695} C_VEL
LIN {X 0,Y 559.136,Z 133.832,A -85,B 0,C 180,E1 -2777.662,E2 -2777.662} C_VEL
LIN {X 0,Y 559.114,Z 133.837,A -85,B 0,C 180,E1 -2779.865,E2 -2779.865} C_VEL
LIN {X 0,Y 559.145,Z 133.832,A -85,B 0,C 180,E1 -2782.78,E2 -2782.78} C_VEL
LIN {X 0,Y 559.222,Z 133.821,A -85,B 0,C 180,E1 -2784.953,E2 -2784.953} C_VEL
LIN {X 0,Y 559.245,Z 133.822,A -85,B 0,C 180,E1 -2787.84,E2 -2787.84} C_VEL
LIN {X 0,Y 559.25,Z 133.825,A -85,B 0,C 180,E1 -2790,E2 -2790} C_VEL
LIN {X 0,Y 559.202,Z 133.823,A -85,B 0,C 180,E1 -2792.882,E2 -2792.882} C_VEL
LIN {X 0,Y 559.201,Z 133.83,A -85,B 0,C 180,E1 -2795.77,E2 -2795.77} C_VEL
LIN {X 0,Y 559.147,Z 133.83,A -85,B 0,C 180,E1 -2798.675,E2 -2798.675} C_VEL
LIN {X 0,Y 559.151,Z 133.835,A -85,B 0,C 180,E1 -2801.602,E2 -2801.602} C_VEL
LIN {X 0,Y 559.149,Z 133.83,A -85,B 0,C 180,E1 -2804.576,E2 -2804.576} C_VEL
LIN {X 0,Y 559.108,Z 133.842,A -85,B 0,C 180,E1 -2807.558,E2 -2807.558} C_VEL
LIN {X 0,Y 559.132,Z 133.838,A -85,B 0,C 180,E1 -2809.839,E2 -2809.839} C_VEL
LIN {X 0,Y 559.097,Z 133.838,A -85,B 0,C 180,E1 -2812.154,E2 -2812.154} C_VEL
LIN {X 0,Y 559.134,Z 133.836,A -85,B 0,C 180,E1 -2815.178,E2 -2815.178} C_VEL
LIN {X 0,Y 559.095,Z 133.842,A -85,B 0,C 180,E1 -2817.716,E2 -2817.716} C_VEL
LIN {X 0,Y 559.089,Z 133.837,A -85,B 0,C 180,E1 -2820.186,E2 -2820.186} C_VEL
LIN {X 0,Y 559.141,Z 133.832,A -85,B 0,C 180,E1 -2822.716,E2 -2822.716} C_VEL
LIN {X 0,Y 559.108,Z 133.844,A -85,B 0,C 180,E1 -2825.325,E2 -2825.325} C_VEL
LIN {X 0,Y 559.116,Z 133.834,A -85,B 0,C 180,E1 -2828.018,E2 -2828.018} C_VEL
LIN {X 0,Y 559.143,Z 133.831,A -85,B 0,C 180,E1 -2829.94,E2 -2829.94} C_VEL
LIN {X 0,Y 559.116,Z 133.842,A -85,B 0,C 180,E1 -2833.194,E2 -2833.194} C_VEL
LIN {X 0,Y 559.116,Z 133.834,A -85,B 0,C 180,E1 -2835.764,E2 -2835.764} C_VEL
LIN {X 0,Y 559.093,Z 133.837,A -85,B 0,C 180,E1 -2838.224,E2 -2838.224} C_VEL
LIN {X 0,Y 559.16,Z 133.836,A -85,B 0,C 180,E1 -2841.065,E2 -2841.065} C_VEL
LIN {X 0,Y 559.105,Z 133.835,A -85,B 0,C 180,E1 -2843.787,E2 -2843.787} C_VEL
LIN {X 0,Y 559.136,Z 133.835,A -85,B 0,C 180,E1 -2846.424,E2 -2846.424} C_VEL
LIN {X 0,Y 559.134,Z 133.838,A -85,B 0,C 180,E1 -2848.98,E2 -2848.98} C_VEL
LIN {X 0,Y 559.095,Z 133.836,A -85,B 0,C 180,E1 -2851.632,E2 -2851.632} C_VEL
LIN {X 0,Y 559.145,Z 133.831,A -85,B 0,C 180,E1 -2853.901,E2 -2853.901} C_VEL
LIN {X 0,Y 559.088,Z 133.84,A -85,B 0,C 180,E1 -2857.065,E2 -2857.065} C_VEL
LIN {X 0,Y 559.139,Z 133.831,A -85,B 0,C 180,E1 -2859.394,E2 -2859.394} C_VEL
LIN {X 0,Y 559.105,Z 133.835,A -85,B 0,C 180,E1 -2861.685,E2 -2861.685} C_VEL
LIN {X 0,Y 559.12,Z 133.838,A -85,B 0,C 180,E1 -2864.695,E2 -2864.695} C_VEL
LIN {X 0,Y 559.133,Z 133.833,A -85,B 0,C 180,E1 -2867.662,E2 -2867.662} C_VEL
LIN {X 0,Y 559.111,Z 133.837,A -85,B 0,C 180,E1 -2869.865,E2 -2869.865} C_VEL
LIN {X 0,Y 559.141,Z 133.832,A -85,B 0,C 180,E1 -2872.78,E2 -2872.78} C_VEL
LIN {X 0,Y 559.219,Z 133.821,A -85,B 0,C 180,E1 -2874.953,E2 -2874.953} C_VEL
LIN {X 0,Y 559.243,Z 133.823,A -85,B 0,C 180,E1 -2877.84,E2 -2877.84} C_VEL
LIN {X 0,Y 559.247,Z 133.826,A -85,B 0,C 180,E1 -2880,E2 -2880} C_VEL
LIN {X 0,Y 559.199,Z 133.823,A -85,B 0,C 180,E1 -2882.882,E2 -2882.882} C_VEL
LIN {X 0,Y 559.199,Z 133.83,A -85,B 0,C 180,E1 -2885.771,E2 -2885.771} C_VEL
LIN {X 0,Y 559.144,Z 133.83,A -85,B 0,C 180,E1 -2888.675,E2 -2888.675} C_VEL
LIN {X 0,Y 559.148,Z 133.836,A -85,B 0,C 180,E1 -2891.602,E2 -2891.602} C_VEL
LIN {X 0,Y 559.147,Z 133.83,A -85,B 0,C 180,E1 -2894.577,E2 -2894.577} C_VEL
LIN {X 0,Y 559.106,Z 133.843,A -85,B 0,C 180,E1 -2897.559,E2 -2897.559} C_VEL
LIN {X 0,Y 559.13,Z 133.838,A -85,B 0,C 180,E1 -2899.839,E2 -2899.839} C_VEL
LIN {X 0,Y 559.095,Z 133.838,A -85,B 0,C 180,E1 -2902.155,E2 -2902.155} C_VEL
LIN {X 0,Y 559.134,Z 133.836,A -85,B 0,C 180,E1 -2905.178,E2 -2905.178} C_VEL
LIN {X 0,Y 559.095,Z 133.841,A -85,B 0,C 180,E1 -2907.717,E2 -2907.717} C_VEL
LIN {X 0,Y 559.087,Z 133.837,A -85,B 0,C 180,E1 -2910.187,E2 -2910.187} C_VEL
LIN {X 0,Y 559.142,Z 133.832,A -85,B 0,C 180,E1 -2912.717,E2 -2912.717} C_VEL
LIN {X 0,Y 559.108,Z 133.844,A -85,B 0,C 180,E1 -2915.326,E2 -2915.326} C_VEL
LIN {X 0,Y 559.118,Z 133.834,A -85,B 0,C 180,E1 -2918.019,E2 -2918.019} C_VEL
LIN {X 0,Y 559.098,Z 133.84,A -85,B 0,C 180,E1 -2920.818,E2 -2920.818} C_VEL
LIN {X 0,Y 559.097,Z 133.837,A -85,B 0,C 180,E1 -2923.739,E2 -2923.739} C_VEL
LIN {X 0,Y 559.097,Z 133.836,A -85,B 0,C 180,E1 -2926.262,E2 -2926.262} C_VEL
LIN {X 0,Y 559.1,Z 133.842,A -85,B 0,C 180,E1 -2929.183,E2 -2929.183} C_VEL
LIN {X 0,Y 559.12,Z 133.833,A -85,B 0,C 180,E1 -2931.982,E2 -2931.982} C_VEL
LIN {X 0,Y 559.114,Z 133.843,A -85,B 0,C 180,E1 -2934.79,E2 -2934.79} C_VEL
LIN {X 0,Y 559.134,Z 133.833,A -85,B 0,C 180,E1 -2937.369,E2 -2937.369} C_VEL
LIN {X 0,Y 559.095,Z 133.838,A -85,B 0,C 180,E1 -2940.153,E2 -2940.153} C_VEL
LIN {X 0,Y 559.11,Z 133.837,A -85,B 0,C 180,E1 -2943.186,E2 -2943.186} C_VEL
LIN {X 0,Y 559.09,Z 133.839,A -85,B 0,C 180,E1 -2945.492,E2 -2945.492} C_VEL
LIN {X 0,Y 559.137,Z 133.979,A -85,B 0,C 180,E1 -2946.695,E2 -2946.695} C_VEL
LIN {X 0,Y 560.003,Z 140.248,A -85,B 0,C 180,E1 -2947.689,E2 -2947.689} C_VEL
LIN {X 0,Y 559.795,Z 156.791,A -85,B 0,C 180,E1 -2950.186,E2 -2950.186} C_VEL
LIN {X 0,Y 559.546,Z 175.268,A -85,B 0,C 180,E1 -2952.935,E2 -2952.935} C_VEL
LIN {X 0,Y 559.388,Z 194.941,A -85,B 0,C 180,E1 -2955.819,E2 -2955.819} C_VEL
LIN {X 0,Y 560.271,Z 202.156,A -85,B 0,C 180,E1 -2955.934,E2 -2955.934} C_VEL
LIN {X 0,Y 560.073,Z 302.949,A -85,B 0,C 180,E1 -2957.246,E2 -2957.246} C_VEL
LIN {X 0,Y 559.916,Z 316.219,A -85,B 0,C 180,E1 -2957.564,E2 -2957.564} C_VEL
LIN {X 0,Y 559.792,Z 328.378,A -85,B 0,C 180,E1 -2957.999,E2 -2957.999} C_VEL
LIN {X 0,Y 559.629,Z 340.194,A -85,B 0,C 180,E1 -2958.567,E2 -2958.567} C_VEL
LIN {X 0,Y 559.458,Z 352.194,A -85,B 0,C 180,E1 -2959.322,E2 -2959.322} C_VEL
LIN {X 0,Y 559.305,Z 362.605,A -85,B 0,C 180,E1 -2960.142,E2 -2960.142} C_VEL
LIN {X 0,Y 559.162,Z 371.113,A -85,B 0,C 180,E1 -2960.961,E2 -2960.961} C_VEL
LIN {X 0,Y 559.05,Z 378.961,A -85,B 0,C 180,E1 -2961.87,E2 -2961.87} C_VEL
LIN {X 0,Y 558.944,Z 386.623,A -85,B 0,C 180,E1 -2962.958,E2 -2962.958} C_VEL
LIN {X 0,Y 558.936,Z 393.679,A -85,B 0,C 180,E1 -2964.227,E2 -2964.227} C_VEL
LIN {X 0,Y 558.826,Z 398.373,A -85,B 0,C 180,E1 -2965.311,E2 -2965.311} C_VEL
LIN {X 0,Y 558.836,Z 401.958,A -85,B 0,C 180,E1 -2966.395,E2 -2966.395} C_VEL
LIN {X 0,Y 558.799,Z 403.807,A -85,B 0,C 180,E1 -2967.116,E2 -2967.116} C_VEL
LIN {X 0,Y 558.745,Z 406.183,A -85,B 0,C 180,E1 -2968.558,E2 -2968.558} C_VEL
LIN {X 0,Y 558.74,Z 407,A -85,B 0,C 180,E1 -2970,E2 -2970} C_VEL
LIN {X 0,Y 558.745,Z 406.184,A -85,B 0,C 180,E1 -2971.441,E2 -2971.441} C_VEL
LIN {X 0,Y 558.799,Z 403.81,A -85,B 0,C 180,E1 -2972.883,E2 -2972.883} C_VEL
LIN {X 0,Y 558.844,Z 400.896,A -85,B 0,C 180,E1 -2973.966,E2 -2973.966} C_VEL
LIN {X 0,Y 558.798,Z 396.949,A -85,B 0,C 180,E1 -2975.051,E2 -2975.051} C_VEL
LIN {X 0,Y 558.919,Z 391.868,A -85,B 0,C 180,E1 -2976.135,E2 -2976.135} C_VEL
LIN {X 0,Y 558.977,Z 385.468,A -85,B 0,C 180,E1 -2977.223,E2 -2977.223} C_VEL
LIN {X 0,Y 559.099,Z 377.479,A -85,B 0,C 180,E1 -2978.311,E2 -2978.311} C_VEL
LIN {X 0,Y 559.194,Z 369.336,A -85,B 0,C 180,E1 -2979.221,E2 -2979.221} C_VEL
LIN {X 0,Y 559.357,Z 359.4,A -85,B 0,C 180,E1 -2980.131,E2 -2980.131} C_VEL
LIN {X 0,Y 559.556,Z 348.401,A -85,B 0,C 180,E1 -2980.936,E2 -2980.936} C_VEL
LIN {X 0,Y 559.671,Z 336.462,A -85,B 0,C 180,E1 -2981.627,E2 -2981.627} C_VEL
LIN {X 0,Y 559.821,Z 324.983,A -85,B 0,C 180,E1 -2982.138,E2 -2982.138} C_VEL
LIN {X 0,Y 559.981,Z 312.185,A -85,B 0,C 180,E1 -2982.549,E2 -2982.549} C_VEL
LIN {X 0,Y 560.088,Z 298.613,A -85,B 0,C 180,E1 -2982.823,E2 -2982.823} C_VEL
LIN {X 0,Y 560.2,Z 200.578,A -85,B 0,C 180,E1 -2984.087,E2 -2984.087} C_VEL
LIN {X 0,Y 559.37,Z 194.668,A -85,B 0,C 180,E1 -2984.205,E2 -2984.205} C_VEL
LIN {X 0,Y 559.525,Z 175.128,A -85,B 0,C 180,E1 -2987.063,E2 -2987.063} C_VEL
LIN {X 0,Y 559.714,Z 159.567,A -85,B 0,C 180,E1 -2989.361,E2 -2989.361} C_VEL
LIN {X 0,Y 559.973,Z 142.687,A -85,B 0,C 180,E1 -2991.882,E2 -2991.882} C_VEL
LIN {X 0,Y 559.711,Z 137.231,A -85,B 0,C 180,E1 -2992.712,E2 -2992.712} C_VEL
LIN {X 0,Y 559.118,Z 133.843,A -85,B 0,C 180,E1 -2993.276,E2 -2993.276} C_VEL
LIN {X 0,Y 559.139,Z 133.834,A -85,B 0,C 180,E1 -2996.099,E2 -2996.099} C_VEL
LIN {X 0,Y 559.096,Z 133.839,A -85,B 0,C 180,E1 -2998.533,E2 -2998.533} C_VEL
LIN {X 0,Y 559.116,Z 133.845,A -85,B 0,C 180,E1 -3001.267,E2 -3001.267} C_VEL
LIN {X 0,Y 559.148,Z 133.831,A -85,B 0,C 180,E1 -3003.946,E2 -3003.946} C_VEL
LIN {X 0,Y 559.113,Z 133.844,A -85,B 0,C 180,E1 -3007.11,E2 -3007.11} C_VEL
LIN {X 0,Y 559.143,Z 133.832,A -85,B 0,C 180,E1 -3009.868,E2 -3009.868} C_VEL
LIN {X 0,Y 559.109,Z 133.841,A -85,B 0,C 180,E1 -3012.747,E2 -3012.747} C_VEL
LIN {X 0,Y 559.118,Z 133.834,A -85,B 0,C 180,E1 -3015.763,E2 -3015.763} C_VEL
LIN {X 0,Y 559.093,Z 133.837,A -85,B 0,C 180,E1 -3018.223,E2 -3018.223} C_VEL
LIN {X 0,Y 559.161,Z 133.832,A -85,B 0,C 180,E1 -3021.192,E2 -3021.192} C_VEL
LIN {X 0,Y 559.106,Z 133.834,A -85,B 0,C 180,E1 -3023.786,E2 -3023.786} C_VEL
LIN {X 0,Y 559.137,Z 133.836,A -85,B 0,C 180,E1 -3026.423,E2 -3026.423} C_VEL
LIN {X 0,Y 559.13,Z 133.836,A -85,B 0,C 180,E1 -3028.979,E2 -3028.979} C_VEL
LIN {X 0,Y 559.095,Z 133.836,A -85,B 0,C 180,E1 -3031.631,E2 -3031.631} C_VEL
LIN {X 0,Y 559.145,Z 133.83,A -85,B 0,C 180,E1 -3033.901,E2 -3033.901} C_VEL
LIN {X 0,Y 559.089,Z 133.844,A -85,B 0,C 180,E1 -3036.582,E2 -3036.582} C_VEL
LIN {X 0,Y 559.104,Z 133.836,A -85,B 0,C 180,E1 -3039.392,E2 -3039.392} C_VEL
LIN {X 0,Y 559.099,Z 133.836,A -85,B 0,C 180,E1 -3041.684,E2 -3041.684} C_VEL
LIN {X 0,Y 559.119,Z 133.836,A -85,B 0,C 180,E1 -3044.694,E2 -3044.694} C_VEL
LIN {X 0,Y 559.136,Z 133.833,A -85,B 0,C 180,E1 -3047.662,E2 -3047.662} C_VEL
LIN {X 0,Y 559.112,Z 133.839,A -85,B 0,C 180,E1 -3049.864,E2 -3049.864} C_VEL
LIN {X 0,Y 559.139,Z 133.832,A -85,B 0,C 180,E1 -3052.779,E2 -3052.779} C_VEL
LIN {X 0,Y 559.217,Z 133.82,A -85,B 0,C 180,E1 -3054.953,E2 -3054.953} C_VEL
LIN {X 0,Y 559.242,Z 133.826,A -85,B 0,C 180,E1 -3057.839,E2 -3057.839} C_VEL
LIN {X 0,Y 559.245,Z 133.826,A -85,B 0,C 180,E1 -3060,E2 -3060} C_VEL
LIN {X 0,Y 559.197,Z 133.824,A -85,B 0,C 180,E1 -3062.881,E2 -3062.881} C_VEL
LIN {X 0,Y 559.198,Z 133.832,A -85,B 0,C 180,E1 -3065.77,E2 -3065.77} C_VEL
LIN {X 0,Y 559.142,Z 133.832,A -85,B 0,C 180,E1 -3068.675,E2 -3068.675} C_VEL
LIN {X 0,Y 559.146,Z 133.84,A -85,B 0,C 180,E1 -3071.601,E2 -3071.601} C_VEL
LIN {X 0,Y 559.149,Z 133.832,A -85,B 0,C 180,E1 -3074.579,E2 -3074.579} C_VEL
LIN {X 0,Y 559.098,Z 133.846,A -85,B 0,C 180,E1 -3077.559,E2 -3077.559} C_VEL
LIN {X 0,Y 559.143,Z 133.837,A -85,B 0,C 180,E1 -3079.838,E2 -3079.838} C_VEL
LIN {X 0,Y 559.094,Z 133.84,A -85,B 0,C 180,E1 -3082.154,E2 -3082.154} C_VEL
LIN {X 0,Y 559.149,Z 133.974,A -85,B 0,C 180,E1 -3084.209,E2 -3084.209} C_VEL
LIN {X 0,Y 559.494,Z 138.848,A -85,B 0,C 180,E1 -3085.06,E2 -3085.06} C_VEL
LIN {X 0,Y 559.352,Z 154.007,A -85,B 0,C 180,E1 -3087.703,E2 -3087.703} C_VEL
LIN {X 0,Y 559.328,Z 160.192,A -85,B 0,C 180,E1 -3088.789,E2 -3088.789} C_VEL
LIN {X 0,Y 559.043,Z 162.53,A -85,B 0,C 180,E1 -3089.101,E2 -3089.101} C_VEL
LIN {X 0,Y 557.92,Z 167.092,A -85,B 0,C 180,E1 -3089.457,E2 -3089.457} C_VEL
LIN {X 0,Y 556.411,Z 172.329,A -85,B 0,C 180,E1 -3089.694,E2 -3089.694} C_VEL
LIN {X 0,Y 554.38,Z 180.164,A -85,B 0,C 180,E1 -3089.89,E2 -3089.89} C_VEL
LIN {X 0,Y 553.466,Z 186.258,A -85,B 0,C 180,E1 -3089.982,E2 -3089.982} C_VEL
LIN {X 0,Y 553.367,Z 188.315,A -85,B 0,C 180,E1 -3090.009,E2 -3090.009} C_VEL
LIN {X 0,Y 553.108,Z 273.74,A -85,B 0,C 180,E1 -3091.144,E2 -3091.144} C_VEL
LIN {X 0,Y 552.972,Z 286.116,A -85,B 0,C 180,E1 -3091.452,E2 -3091.452} C_VEL
LIN {X 0,Y 552.858,Z 296.612,A -85,B 0,C 180,E1 -3091.82,E2 -3091.82} C_VEL
LIN {X 0,Y 552.681,Z 307.739,A -85,B 0,C 180,E1 -3092.332,E2 -3092.332} C_VEL
LIN {X 0,Y 552.463,Z 320.208,A -85,B 0,C 180,E1 -3093.082,E2 -3093.082} C_VEL
LIN {X 0,Y 552.291,Z 329.961,A -85,B 0,C 180,E1 -3093.829,E2 -3093.829} C_VEL
LIN {X 0,Y 552.19,Z 338.661,A -85,B 0,C 180,E1 -3094.636,E2 -3094.636} C_VEL
LIN {X 0,Y 552.036,Z 345.908,A -85,B 0,C 180,E1 -3095.435,E2 -3095.435} C_VEL
LIN {X 0,Y 551.919,Z 352.218,A -85,B 0,C 180,E1 -3096.255,E2 -3096.255} C_VEL
LIN {X 0,Y 551.861,Z 358.436,A -85,B 0,C 180,E1 -3097.222,E2 -3097.222} C_VEL
LIN {X 0,Y 551.803,Z 363.637,A -85,B 0,C 180,E1 -3098.204,E2 -3098.204} C_VEL
LIN {X 0,Y 551.739,Z 368.178,A -85,B 0,C 180,E1 -3099.264,E2 -3099.264} C_VEL
LIN {X 0,Y 551.703,Z 372.254,A -85,B 0,C 180,E1 -3100.517,E2 -3100.517} C_VEL
LIN {X 0,Y 551.679,Z 374.48,A -85,B 0,C 180,E1 -3101.486,E2 -3101.486} C_VEL
LIN {X 0,Y 551.649,Z 375.997,A -85,B 0,C 180,E1 -3102.471,E2 -3102.471} C_VEL
LIN {X 0,Y 551.663,Z 376.793,A -85,B 0,C 180,E1 -3103.467,E2 -3103.467} C_VEL
LIN {X 0,Y 551.697,Z 376.846,A -85,B 0,C 180,E1 -3104.491,E2 -3104.491} C_VEL
LIN {X 0,Y 551.698,Z 376.112,A -85,B 0,C 180,E1 -3105.523,E2 -3105.523} C_VEL
LIN {X 0,Y 551.672,Z 373.565,A -85,B 0,C 180,E1 -3107.051,E2 -3107.051} C_VEL
LIN {X 0,Y 551.742,Z 369.339,A -85,B 0,C 180,E1 -3108.52,E2 -3108.52} C_VEL
LIN {X 0,Y 551.774,Z 363.869,A -85,B 0,C 180,E1 -3109.838,E2 -3109.838} C_VEL
LIN {X 0,Y 551.866,Z 359.193,A -85,B 0,C 180,E1 -3110.736,E2 -3110.736} C_VEL
LIN {X 0,Y 551.886,Z 353.904,A -85,B 0,C 180,E1 -3111.59,E2 -3111.59} C_VEL
LIN {X 0,Y 551.992,Z 348.578,A -85,B 0,C 180,E1 -3112.329,E2 -3112.329} C_VEL
LIN {X 0,Y 552.118,Z 340.588,A -85,B 0,C 180,E1 -3113.255,E2 -3113.255} C_VEL
LIN {X 0,Y 552.29,Z 332.246,A -85,B 0,C 180,E1 -3114.06,E2 -3114.06} C_VEL
LIN {X 0,Y 552.443,Z 323.218,A -85,B 0,C 180,E1 -3114.786,E2 -3114.786} C_VEL
LIN {X 0,Y 552.565,Z 314.69,A -85,B 0,C 180,E1 -3115.358,E2 -3115.358} C_VEL
LIN {X 0,Y 552.719,Z 304.86,A -85,B 0,C 180,E1 -3115.9,E2 -3115.9} C_VEL
LIN {X 0,Y 552.861,Z 295.334,A -85,B 0,C 180,E1 -3116.32,E2 -3116.32} C_VEL
LIN {X 0,Y 553.002,Z 284.534,A -85,B 0,C 180,E1 -3116.685,E2 -3116.685} C_VEL
LIN {X 0,Y 553.125,Z 272.956,A -85,B 0,C 180,E1 -3116.96,E2 -3116.96} C_VEL
LIN {X 0,Y 553.345,Z 172.775,A -85,B 0,C 180,E1 -3118.288,E2 -3118.288} C_VEL
LIN {X 0,Y 552.252,Z 166.447,A -85,B 0,C 180,E1 -3118.403,E2 -3118.403} C_VEL
LIN {X 0,Y 552.444,Z 149.936,A -85,B 0,C 180,E1 -3121.377,E2 -3121.377} C_VEL
LIN {X 0,Y 552.605,Z 137.848,A -85,B 0,C 180,E1 -3123.569,E2 -3123.569} C_VEL
LIN {X 0,Y 552.104,Z 134.716,A -85,B 0,C 180,E1 -3124.178,E2 -3124.178} C_VEL
LIN {X 0,Y 552.04,Z 134.724,A -85,B 0,C 180,E1 -3126.756,E2 -3126.756} C_VEL
LIN {X 0,Y 552.09,Z 134.712,A -85,B 0,C 180,E1 -3129.119,E2 -3129.119} C_VEL
LIN {X 0,Y 552.071,Z 134.711,A -85,B 0,C 180,E1 -3131.443,E2 -3131.443} C_VEL
LIN {X 0,Y 552.067,Z 134.712,A -85,B 0,C 180,E1 -3133.736,E2 -3133.736} C_VEL
LIN {X 0,Y 552.105,Z 134.711,A -85,B 0,C 180,E1 -3136.004,E2 -3136.004} C_VEL
LIN {X 0,Y 552.121,Z 134.706,A -85,B 0,C 180,E1 -3138.993,E2 -3138.993} C_VEL
LIN {X 0,Y 552.104,Z 134.712,A -85,B 0,C 180,E1 -3141.951,E2 -3141.951} C_VEL
LIN {X 0,Y 552.199,Z 134.696,A -85,B 0,C 180,E1 -3144.889,E2 -3144.889} C_VEL
LIN {X 0,Y 552.216,Z 134.698,A -85,B 0,C 180,E1 -3147.812,E2 -3147.812} C_VEL
LIN {X 0,Y 552.219,Z 134.701,A -85,B 0,C 180,E1 -3150,E2 -3150} C_VEL
LIN {X 0,Y 552.17,Z 134.699,A -85,B 0,C 180,E1 -3152.918,E2 -3152.918} C_VEL
LIN {X 0,Y 552.17,Z 134.707,A -85,B 0,C 180,E1 -3155.844,E2 -3155.844} C_VEL
LIN {X 0,Y 552.12,Z 134.705,A -85,B 0,C 180,E1 -3158.786,E2 -3158.786} C_VEL
LIN {X 0,Y 552.096,Z 134.717,A -85,B 0,C 180,E1 -3161.752,E2 -3161.752} C_VEL
LIN {X 0,Y 552.115,Z 134.706,A -85,B 0,C 180,E1 -3164.749,E2 -3164.749} C_VEL
LIN {X 0,Y 552.07,Z 134.719,A -85,B 0,C 180,E1 -3167.79,E2 -3167.79} C_VEL
LIN {X 0,Y 552.087,Z 134.712,A -85,B 0,C 180,E1 -3170.103,E2 -3170.103} C_VEL
LIN {X 0,Y 552.037,Z 134.716,A -85,B 0,C 180,E1 -3172.453,E2 -3172.453} C_VEL
LIN {X 0,Y 552.078,Z 134.717,A -85,B 0,C 180,E1 -3175.334,E2 -3175.334} C_VEL
LIN {X 0,Y 552.043,Z 134.716,A -85,B 0,C 180,E1 -3178.102,E2 -3178.102} C_VEL
LIN {X 0,Y 552.065,Z 134.712,A -85,B 0,C 180,E1 -3180.611,E2 -3180.611} C_VEL
LIN {X 0,Y 552.097,Z 134.715,A -85,B 0,C 180,E1 -3183.187,E2 -3183.187} C_VEL
LIN {X 0,Y 552.063,Z 134.714,A -85,B 0,C 180,E1 -3185.845,E2 -3185.845} C_VEL
LIN {X 0,Y 552.104,Z 134.708,A -85,B 0,C 180,E1 -3188.59,E2 -3188.59} C_VEL
LIN {X 0,Y 552.052,Z 134.719,A -85,B 0,C 180,E1 -3191.452,E2 -3191.452} C_VEL
LIN {X 0,Y 552.068,Z 134.714,A -85,B 0,C 180,E1 -3194.529,E2 -3194.529} C_VEL
LIN {X 0,Y 552.076,Z 134.712,A -85,B 0,C 180,E1 -3197.59,E2 -3197.59} C_VEL
LIN {X 0,Y 552.117,Z 134.708,A -85,B 0,C 180,E1 -3200.472,E2 -3200.472} C_VEL
LIN {X 0,Y 552.062,Z 134.715,A -85,B 0,C 180,E1 -3203.322,E2 -3203.322} C_VEL
LIN {X 0,Y 552.088,Z 134.709,A -85,B 0,C 180,E1 -3205.937,E2 -3205.937} C_VEL
LIN {X 0,Y 552.096,Z 134.714,A -85,B 0,C 180,E1 -3208.54,E2 -3208.54} C_VEL
LIN {X 0,Y 552.063,Z 134.713,A -85,B 0,C 180,E1 -3211.448,E2 -3211.448} C_VEL
LIN {X 0,Y 552.073,Z 134.716,A -85,B 0,C 180,E1 -3214.353,E2 -3214.353} C_VEL
LIN {X 0,Y 552.043,Z 134.722,A -85,B 0,C 180,E1 -3216.756,E2 -3216.756} C_VEL
LIN {X 0,Y 552.087,Z 134.711,A -85,B 0,C 180,E1 -3219.119,E2 -3219.119} C_VEL
LIN {X 0,Y 552.068,Z 134.712,A -85,B 0,C 180,E1 -3221.443,E2 -3221.443} C_VEL
LIN {X 0,Y 552.064,Z 134.713,A -85,B 0,C 180,E1 -3223.736,E2 -3223.736} C_VEL
LIN {X 0,Y 552.101,Z 134.711,A -85,B 0,C 180,E1 -3226.004,E2 -3226.004} C_VEL
LIN {X 0,Y 552.118,Z 134.706,A -85,B 0,C 180,E1 -3228.993,E2 -3228.993} C_VEL
LIN {X 0,Y 552.101,Z 134.712,A -85,B 0,C 180,E1 -3231.951,E2 -3231.951} C_VEL
LIN {X 0,Y 552.196,Z 134.696,A -85,B 0,C 180,E1 -3234.889,E2 -3234.889} C_VEL
LIN {X 0,Y 552.213,Z 134.698,A -85,B 0,C 180,E1 -3237.812,E2 -3237.812} C_VEL
LIN {X 0,Y 552.216,Z 134.702,A -85,B 0,C 180,E1 -3240,E2 -3240} C_VEL
LIN {X 0,Y 552.167,Z 134.699,A -85,B 0,C 180,E1 -3242.919,E2 -3242.919} C_VEL
LIN {X 0,Y 552.168,Z 134.707,A -85,B 0,C 180,E1 -3245.845,E2 -3245.845} C_VEL
LIN {X 0,Y 552.117,Z 134.705,A -85,B 0,C 180,E1 -3248.787,E2 -3248.787} C_VEL
LIN {X 0,Y 552.093,Z 134.718,A -85,B 0,C 180,E1 -3251.752,E2 -3251.752} C_VEL
LIN {X 0,Y 552.113,Z 134.706,A -85,B 0,C 180,E1 -3254.749,E2 -3254.749} C_VEL
LIN {X 0,Y 552.068,Z 134.719,A -85,B 0,C 180,E1 -3257.79,E2 -3257.79} C_VEL
LIN {X 0,Y 552.086,Z 134.712,A -85,B 0,C 180,E1 -3260.103,E2 -3260.103} C_VEL
LIN {X 0,Y 552.035,Z 134.716,A -85,B 0,C 180,E1 -3262.454,E2 -3262.454} C_VEL
LIN {X 0,Y 552.077,Z 134.718,A -85,B 0,C 180,E1 -3265.334,E2 -3265.334} C_VEL
LIN {X 0,Y 552.043,Z 134.716,A -85,B 0,C 180,E1 -3268.102,E2 -3268.102} C_VEL
LIN {X 0,Y 552.063,Z 134.713,A -85,B 0,C 180,E1 -3270.612,E2 -3270.612} C_VEL
LIN {X 0,Y 552.098,Z 134.715,A -85,B 0,C 180,E1 -3273.187,E2 -3273.187} C_VEL
LIN {X 0,Y 552.062,Z 134.714,A -85,B 0,C 180,E1 -3275.846,E2 -3275.846} C_VEL
LIN {X 0,Y 552.105,Z 134.708,A -85,B 0,C 180,E1 -3278.59,E2 -3278.59} C_VEL
LIN {X 0,Y 552.052,Z 134.718,A -85,B 0,C 180,E1 -3281.453,E2 -3281.453} C_VEL
LIN {X 0,Y 552.071,Z 134.713,A -85,B 0,C 180,E1 -3284.53,E2 -3284.53} C_VEL
LIN {X 0,Y 552.078,Z 134.712,A -85,B 0,C 180,E1 -3287.591,E2 -3287.591} C_VEL
LIN {X 0,Y 552.09,Z 134.712,A -85,B 0,C 180,E1 -3290.47,E2 -3290.47} C_VEL
LIN {X 0,Y 552.051,Z 134.717,A -85,B 0,C 180,E1 -3293.325,E2 -3293.325} C_VEL
LIN {X 0,Y 552.093,Z 134.709,A -85,B 0,C 180,E1 -3295.937,E2 -3295.937} C_VEL
LIN {X 0,Y 552.079,Z 134.716,A -85,B 0,C 180,E1 -3298.538,E2 -3298.538} C_VEL
LIN {X 0,Y 552.07,Z 134.713,A -85,B 0,C 180,E1 -3301.449,E2 -3301.449} C_VEL
LIN {X 0,Y 552.061,Z 134.718,A -85,B 0,C 180,E1 -3304.353,E2 -3304.353} C_VEL
LIN {X 0,Y 552.094,Z 134.904,A -85,B 0,C 180,E1 -3306.548,E2 -3306.548} C_VEL
LIN {X 0,Y 553.05,Z 141.349,A -85,B 0,C 180,E1 -3307.59,E2 -3307.59} C_VEL
LIN {X 0,Y 552.863,Z 156.622,A -85,B 0,C 180,E1 -3309.927,E2 -3309.927} C_VEL
LIN {X 0,Y 552.557,Z 174.743,A -85,B 0,C 180,E1 -3312.659,E2 -3312.659} C_VEL
LIN {X 0,Y 552.353,Z 194.663,A -85,B 0,C 180,E1 -3315.628,E2 -3315.628} C_VEL
LIN {X 0,Y 553.381,Z 202.38,A -85,B 0,C 180,E1 -3315.763,E2 -3315.763} C_VEL
LIN {X 0,Y 553.133,Z 302.537,A -85,B 0,C 180,E1 -3317.083,E2 -3317.083} C_VEL
LIN {X 0,Y 552.981,Z 315.909,A -85,B 0,C 180,E1 -3317.406,E2 -3317.406} C_VEL
LIN {X 0,Y 552.847,Z 328.128,A -85,B 0,C 180,E1 -3317.846,E2 -3317.846} C_VEL
LIN {X 0,Y 552.654,Z 338.998,A -85,B 0,C 180,E1 -3318.366,E2 -3318.366} C_VEL
LIN {X 0,Y 552.479,Z 350.773,A -85,B 0,C 180,E1 -3319.093,E2 -3319.093} C_VEL
LIN {X 0,Y 552.298,Z 361.458,A -85,B 0,C 180,E1 -3319.923,E2 -3319.923} C_VEL
LIN {X 0,Y 552.131,Z 371.082,A -85,B 0,C 180,E1 -3320.845,E2 -3320.845} C_VEL
LIN {X 0,Y 552.013,Z 378.961,A -85,B 0,C 180,E1 -3321.765,E2 -3321.765} C_VEL
LIN {X 0,Y 551.89,Z 386.621,A -85,B 0,C 180,E1 -3322.868,E2 -3322.868} C_VEL
LIN {X 0,Y 551.867,Z 393.679,A -85,B 0,C 180,E1 -3324.153,E2 -3324.153} C_VEL
LIN {X 0,Y 551.725,Z 398.373,A -85,B 0,C 180,E1 -3325.251,E2 -3325.251} C_VEL
LIN {X 0,Y 551.75,Z 401.958,A -85,B 0,C 180,E1 -3326.348,E2 -3326.348} C_VEL
LIN {X 0,Y 551.724,Z 403.806,A -85,B 0,C 180,E1 -3327.079,E2 -3327.079} C_VEL
LIN {X 0,Y 551.645,Z 406.182,A -85,B 0,C 180,E1 -3328.54,E2 -3328.54} C_VEL
LIN {X 0,Y 551.64,Z 407,A -85,B 0,C 180,E1 -3330,E2 -3330} C_VEL
LIN {X 0,Y 551.645,Z 406.184,A -85,B 0,C 180,E1 -3331.46,E2 -3331.46} C_VEL
LIN {X 0,Y 551.723,Z 403.81,A -85,B 0,C 180,E1 -3332.92,E2 -3332.92} C_VEL
LIN {X 0,Y 551.764,Z 400.896,A -85,B 0,C 180,E1 -3334.017,E2 -3334.017} C_VEL
LIN {X 0,Y 551.723,Z 396.949,A -85,B 0,C 180,E1 -3335.116,E2 -3335.116} C_VEL
LIN {X 0,Y 551.801,Z 391.2,A -85,B 0,C 180,E1 -3336.339,E2 -3336.339} C_VEL
LIN {X 0,Y 551.926,Z 384.236,A -85,B 0,C 180,E1 -3337.499,E2 -3337.499} C_VEL
LIN {X 0,Y 552.082,Z 375.988,A -85,B 0,C 180,E1 -3338.602,E2 -3338.602} C_VEL
LIN {X 0,Y 552.2,Z 367.491,A -85,B 0,C 180,E1 -3339.523,E2 -3339.523} C_VEL
LIN {X 0,Y 552.428,Z 356.988,A -85,B 0,C 180,E1 -3340.445,E2 -3340.445} C_VEL
LIN {X 0,Y 552.575,Z 346.126,A -85,B 0,C 180,E1 -3341.214,E2 -3341.214} C_VEL
LIN {X 0,Y 552.751,Z 335.187,A -85,B 0,C 180,E1 -3341.831,E2 -3341.831} C_VEL
LIN {X 0,Y 552.898,Z 323.469,A -85,B 0,C 180,E1 -3342.339,E2 -3342.339} C_VEL
LIN {X 0,Y 553.038,Z 310.875,A -85,B 0,C 180,E1 -3342.732,E2 -3342.732} C_VEL
LIN {X 0,Y 553.16,Z 298.069,A -85,B 0,C 180,E1 -3342.986,E2 -3342.986} C_VEL
LIN {X 0,Y 553.212,Z 200.607,A -85,B 0,C 180,E1 -3344.262,E2 -3344.262} C_VEL
LIN {X 0,Y 552.347,Z 194.531,A -85,B 0,C 180,E1 -3344.375,E2 -3344.375} C_VEL
LIN {X 0,Y 552.541,Z 174.539,A -85,B 0,C 180,E1 -3347.336,E2 -3347.336} C_VEL
LIN {X 0,Y 552.825,Z 156.262,A -85,B 0,C 180,E1 -3350.074,E2 -3350.074} C_VEL
LIN {X 0,Y 552.999,Z 140.835,A -85,B 0,C 180,E1 -3352.412,E2 -3352.412} C_VEL
LIN {X 0,Y 552.062,Z 134.722,A -85,B 0,C 180,E1 -3353.393,E2 -3353.393} C_VEL
LIN {X 0,Y 552.068,Z 134.714,A -85,B 0,C 180,E1 -3356.459,E2 -3356.459} C_VEL
LIN {X 0,Y 552.035,Z 134.722,A -85,B 0,C 180,E1 -3358.932,E2 -3358.932} C_VEL
LIN {X 0,Y 552.09,Z 134.717,A -85,B 0,C 180,E1 -3361.471,E2 -3361.471} C_VEL
LIN {X 0,Y 552.09,Z 134.71,A -85,B 0,C 180,E1 -3364.163,E2 -3364.163} C_VEL
LIN {X 0,Y 552.05,Z 134.719,A -85,B 0,C 180,E1 -3366.751,E2 -3366.751} C_VEL
LIN {X 0,Y 552.088,Z 134.714,A -85,B 0,C 180,E1 -3369.53,E2 -3369.53} C_VEL
LIN {X 0,Y 552.076,Z 134.714,A -85,B 0,C 180,E1 -3372.43,E2 -3372.43} C_VEL
LIN {X 0,Y 552.069,Z 134.714,A -85,B 0,C 180,E1 -3375.559,E2 -3375.559} C_VEL
LIN {X 0,Y 552.05,Z 134.718,A -85,B 0,C 180,E1 -3378.547,E2 -3378.547} C_VEL
LIN {X 0,Y 552.104,Z 134.709,A -85,B 0,C 180,E1 -3381.41,E2 -3381.41} C_VEL
LIN {X 0,Y 552.054,Z 134.719,A -85,B 0,C 180,E1 -3384.562,E2 -3384.562} C_VEL
LIN {X 0,Y 552.099,Z 134.71,A -85,B 0,C 180,E1 -3387.155,E2 -3387.155} C_VEL
LIN {X 0,Y 552.061,Z 134.713,A -85,B 0,C 180,E1 -3389.958,E2 -3389.958} C_VEL
LIN {X 0,Y 552.07,Z 134.713,A -85,B 0,C 180,E1 -3393.012,E2 -3393.012} C_VEL
LIN {X 0,Y 552.064,Z 134.715,A -85,B 0,C 180,E1 -3395.96,E2 -3395.96} C_VEL
LIN {X 0,Y 552.062,Z 134.714,A -85,B 0,C 180,E1 -3399.117,E2 -3399.117} C_VEL
LIN {X 0,Y 552.059,Z 134.712,A -85,B 0,C 180,E1 -3401.442,E2 -3401.442} C_VEL
LIN {X 0,Y 552.064,Z 134.714,A -85,B 0,C 180,E1 -3403.735,E2 -3403.735} C_VEL
LIN {X 0,Y 552.095,Z 134.713,A -85,B 0,C 180,E1 -3406.003,E2 -3406.003} C_VEL
LIN {X 0,Y 552.118,Z 134.706,A -85,B 0,C 180,E1 -3408.992,E2 -3408.992} C_VEL
LIN {X 0,Y 552.099,Z 134.714,A -85,B 0,C 180,E1 -3411.95,E2 -3411.95} C_VEL
LIN {X 0,Y 552.194,Z 134.695,A -85,B 0,C 180,E1 -3414.888,E2 -3414.888} C_VEL
LIN {X 0,Y 552.212,Z 134.701,A -85,B 0,C 180,E1 -3417.812,E2 -3417.812} C_VEL
LIN {X 0,Y 552.214,Z 134.702,A -85,B 0,C 180,E1 -3420,E2 -3420} C_VEL
LIN {X 0,Y 552.165,Z 134.7,A -85,B 0,C 180,E1 -3422.918,E2 -3422.918} C_VEL
LIN {X 0,Y 552.167,Z 134.708,A -85,B 0,C 180,E1 -3425.844,E2 -3425.844} C_VEL
LIN {X 0,Y 552.115,Z 134.707,A -85,B 0,C 180,E1 -3428.786,E2 -3428.786} C_VEL
LIN {X 0,Y 552.092,Z 134.72,A -85,B 0,C 180,E1 -3431.752,E2 -3431.752} C_VEL
LIN {X 0,Y 552.111,Z 134.709,A -85,B 0,C 180,E1 -3434.749,E2 -3434.749} C_VEL
LIN {X 0,Y 552.063,Z 134.719,A -85,B 0,C 180,E1 -3437.79,E2 -3437.79} C_VEL
LIN {X 0,Y 552.101,Z 134.711,A -85,B 0,C 180,E1 -3440.102,E2 -3440.102} C_VEL
LIN {X 0,Y 552.075,Z 134.72,A -85,B 0,C 180,E1 -3443.243,E2 -3443.243} C_VEL
LIN {X 0,Y 552.12,Z 134.914,A -85,B 0,C 180,E1 -3444.137,E2 -3444.137} C_VEL
LIN {X 0,Y 552.501,Z 138.763,A -85,B 0,C 180,E1 -3444.82,E2 -3444.82} C_VEL
LIN {X 0,Y 552.325,Z 153.914,A -85,B 0,C 180,E1 -3447.468,E2 -3447.468} C_VEL
LIN {X 0,Y 552.23,Z 166.315,A -85,B 0,C 180,E1 -3449.679,E2 -3449.679} C_VEL
LIN {X 0,Y 553.446,Z 174.395,A -85,B 0,C 180,E1 -3449.828,E2 -3449.828} C_VEL
LIN {X 0,Y 553.367,Z 188.315,A -85,B 0,C 180,E1 -3450.009,E2 -3450.009} C_VEL
LIN {X 0,Y 552.647,Z 194.159,A -85,B 0,C 180,E1 -3450.067,E2 -3450.067} C_VEL
LIN {X 0,Y 547.043,Z 213.157,A -85,B 0,C 180,E1 -3450.176,E2 -3450.176} C_VEL
LIN {X 0,Y 546.405,Z 218.998,A -85,B 0,C 180,E1 -3450.238,E2 -3450.238} C_VEL
LIN {X 0,Y 546.189,Z 274.296,A -85,B 0,C 180,E1 -3450.99,E2 -3450.99} C_VEL
LIN {X 0,Y 546.024,Z 286.883,A -85,B 0,C 180,E1 -3451.31,E2 -3451.31} C_VEL
LIN {X 0,Y 545.921,Z 298.63,A -85,B 0,C 180,E1 -3451.74,E2 -3451.74} C_VEL
LIN {X 0,Y 545.643,Z 312.181,A -85,B 0,C 180,E1 -3452.421,E2 -3452.421} C_VEL
LIN {X 0,Y 545.427,Z 322.789,A -85,B 0,C 180,E1 -3453.12,E2 -3453.12} C_VEL
LIN {X 0,Y 545.274,Z 332.18,A -85,B 0,C 180,E1 -3453.879,E2 -3453.879} C_VEL
LIN {X 0,Y 545.109,Z 340.354,A -85,B 0,C 180,E1 -3454.673,E2 -3454.673} C_VEL
LIN {X 0,Y 544.983,Z 348.865,A -85,B 0,C 180,E1 -3455.667,E2 -3455.667} C_VEL
LIN {X 0,Y 544.799,Z 357.242,A -85,B 0,C 180,E1 -3456.889,E2 -3456.889} C_VEL
LIN {X 0,Y 544.737,Z 361.853,A -85,B 0,C 180,E1 -3457.71,E2 -3457.71} C_VEL
LIN {X 0,Y 544.696,Z 366.607,A -85,B 0,C 180,E1 -3458.739,E2 -3458.739} C_VEL
LIN {X 0,Y 544.63,Z 370.166,A -85,B 0,C 180,E1 -3459.698,E2 -3459.698} C_VEL
LIN {X 0,Y 544.589,Z 374.027,A -85,B 0,C 180,E1 -3461.159,E2 -3461.159} C_VEL
LIN {X 0,Y 544.558,Z 376.349,A -85,B 0,C 180,E1 -3462.64,E2 -3462.64} C_VEL
LIN {X 0,Y 544.576,Z 377.092,A -85,B 0,C 180,E1 -3464.178,E2 -3464.178} C_VEL
LIN {X 0,Y 544.611,Z 376.616,A -85,B 0,C 180,E1 -3465.214,E2 -3465.214} C_VEL
LIN {X 0,Y 544.571,Z 375.311,A -85,B 0,C 180,E1 -3466.278,E2 -3466.278} C_VEL
LIN {X 0,Y 544.613,Z 373.126,A -85,B 0,C 180,E1 -3467.354,E2 -3467.354} C_VEL
LIN {X 0,Y 544.662,Z 369.958,A -85,B 0,C 180,E1 -3468.451,E2 -3468.451} C_VEL
LIN {X 0,Y 544.681,Z 365.625,A -85,B 0,C 180,E1 -3469.576,E2 -3469.576} C_VEL
LIN {X 0,Y 544.786,Z 359.98,A -85,B 0,C 180,E1 -3470.716,E2 -3470.716} C_VEL
LIN {X 0,Y 544.866,Z 353.67,A -85,B 0,C 180,E1 -3471.748,E2 -3471.748} C_VEL
LIN {X 0,Y 544.986,Z 346.669,A -85,B 0,C 180,E1 -3472.693,E2 -3472.693} C_VEL
LIN {X 0,Y 545.118,Z 340.251,A -85,B 0,C 180,E1 -3473.426,E2 -3473.426} C_VEL
LIN {X 0,Y 545.29,Z 332.559,A -85,B 0,C 180,E1 -3474.175,E2 -3474.175} C_VEL
LIN {X 0,Y 545.46,Z 323.653,A -85,B 0,C 180,E1 -3474.903,E2 -3474.903} C_VEL
LIN {X 0,Y 545.605,Z 314.468,A -85,B 0,C 180,E1 -3475.526,E2 -3475.526} C_VEL
LIN {X 0,Y 545.785,Z 304.011,A -85,B 0,C 180,E1 -3476.102,E2 -3476.102} C_VEL
LIN {X 0,Y 545.994,Z 291.628,A -85,B 0,C 180,E1 -3476.626,E2 -3476.626} C_VEL
LIN {X 0,Y 546.11,Z 277.767,A -85,B 0,C 180,E1 -3477.027,E2 -3477.027} C_VEL
LIN {X 0,Y 546.218,Z 261.757,A -85,B 0,C 180,E1 -3477.29,E2 -3477.29} C_VEL
LIN {X 0,Y 546.509,Z 173.872,A -85,B 0,C 180,E1 -3478.458,E2 -3478.458} C_VEL
LIN {X 0,Y 545.242,Z 166.541,A -85,B 0,C 180,E1 -3478.604,E2 -3478.604} C_VEL
LIN {X 0,Y 545.484,Z 149.302,A -85,B 0,C 180,E1 -3481.74,E2 -3481.74} C_VEL
LIN {X 0,Y 545.641,Z 139.036,A -85,B 0,C 180,E1 -3483.618,E2 -3483.618} C_VEL
LIN {X 0,Y 545.066,Z 135.593,A -85,B 0,C 180,E1 -3484.289,E2 -3484.289} C_VEL
LIN {X 0,Y 544.982,Z 135.597,A -85,B 0,C 180,E1 -3487.24,E2 -3487.24} C_VEL
LIN {X 0,Y 545.097,Z 135.588,A -85,B 0,C 180,E1 -3490.414,E2 -3490.414} C_VEL
LIN {X 0,Y 545.017,Z 135.59,A -85,B 0,C 180,E1 -3493.52,E2 -3493.52} C_VEL
LIN {X 0,Y 545.064,Z 135.586,A -85,B 0,C 180,E1 -3495.819,E2 -3495.819} C_VEL
LIN {X 0,Y 545.067,Z 135.586,A -85,B 0,C 180,E1 -3498.849,E2 -3498.849} C_VEL
LIN {X 0,Y 545.062,Z 135.588,A -85,B 0,C 180,E1 -3501.846,E2 -3501.846} C_VEL
LIN {X 0,Y 545.157,Z 135.574,A -85,B 0,C 180,E1 -3504.823,E2 -3504.823} C_VEL
LIN {X 0,Y 545.187,Z 135.573,A -85,B 0,C 180,E1 -3507.784,E2 -3507.784} C_VEL
LIN {X 0,Y 545.187,Z 135.577,A -85,B 0,C 180,E1 -3510,E2 -3510} C_VEL
LIN {X 0,Y 545.138,Z 135.575,A -85,B 0,C 180,E1 -3512.956,E2 -3512.956} C_VEL
LIN {X 0,Y 545.121,Z 135.586,A -85,B 0,C 180,E1 -3515.92,E2 -3515.92} C_VEL
LIN {X 0,Y 545.063,Z 135.584,A -85,B 0,C 180,E1 -3518.901,E2 -3518.901} C_VEL
LIN {X 0,Y 545.061,Z 135.593,A -85,B 0,C 180,E1 -3521.906,E2 -3521.906} C_VEL
LIN {X 0,Y 545.071,Z 135.584,A -85,B 0,C 180,E1 -3524.944,E2 -3524.944} C_VEL
LIN {X 0,Y 545.038,Z 135.592,A -85,B 0,C 180,E1 -3528.027,E2 -3528.027} C_VEL
LIN {X 0,Y 545.025,Z 135.59,A -85,B 0,C 180,E1 -3530.375,E2 -3530.375} C_VEL
LIN {X 0,Y 544.983,Z 135.594,A -85,B 0,C 180,E1 -3532.76,E2 -3532.76} C_VEL
LIN {X 0,Y 545.03,Z 135.598,A -85,B 0,C 180,E1 -3535.495,E2 -3535.495} C_VEL
LIN {X 0,Y 545.027,Z 135.589,A -85,B 0,C 180,E1 -3538.496,E2 -3538.496} C_VEL
LIN {X 0,Y 545.039,Z 135.592,A -85,B 0,C 180,E1 -3541.676,E2 -3541.676} C_VEL
LIN {X 0,Y 545.039,Z 135.588,A -85,B 0,C 180,E1 -3544.566,E2 -3544.566} C_VEL
LIN {X 0,Y 545.022,Z 135.598,A -85,B 0,C 180,E1 -3547.305,E2 -3547.305} C_VEL
LIN {X 0,Y 545.044,Z 135.587,A -85,B 0,C 180,E1 -3550.144,E2 -3550.144} C_VEL
LIN {X 0,Y 545.01,Z 135.6,A -85,B 0,C 180,E1 -3553.113,E2 -3553.113} C_VEL
LIN {X 0,Y 545.02,Z 135.59,A -85,B 0,C 180,E1 -3556.229,E2 -3556.229} C_VEL
LIN {X 0,Y 545.017,Z 135.598,A -85,B 0,C 180,E1 -3558.88,E2 -3558.88} C_VEL
LIN {X 0,Y 545.036,Z 135.588,A -85,B 0,C 180,E1 -3561.762,E2 -3561.762} C_VEL
LIN {X 0,Y 545.013,Z 135.595,A -85,B 0,C 180,E1 -3564.53,E2 -3564.53} C_VEL
LIN {X 0,Y 545.053,Z 135.589,A -85,B 0,C 180,E1 -3567.211,E2 -3567.211} C_VEL
LIN {X 0,Y 545.014,Z 135.59,A -85,B 0,C 180,E1 -3569.808,E2 -3569.808} C_VEL
LIN {X 0,Y 545.017,Z 135.597,A -85,B 0,C 180,E1 -3572.841,E2 -3572.841} C_VEL
LIN {X 0,Y 545.007,Z 135.591,A -85,B 0,C 180,E1 -3575.629,E2 -3575.629} C_VEL
LIN {X 0,Y 545.026,Z 135.594,A -85,B 0,C 180,E1 -3578.835,E2 -3578.835} C_VEL
LIN {X 0,Y 545.032,Z 135.589,A -85,B 0,C 180,E1 -3581.194,E2 -3581.194} C_VEL
LIN {X 0,Y 545.013,Z 135.59,A -85,B 0,C 180,E1 -3583.52,E2 -3583.52} C_VEL
LIN {X 0,Y 545.06,Z 135.586,A -85,B 0,C 180,E1 -3585.819,E2 -3585.819} C_VEL
LIN {X 0,Y 545.064,Z 135.586,A -85,B 0,C 180,E1 -3588.849,E2 -3588.849} C_VEL
LIN {X 0,Y 545.058,Z 135.588,A -85,B 0,C 180,E1 -3591.846,E2 -3591.846} C_VEL
LIN {X 0,Y 545.154,Z 135.574,A -85,B 0,C 180,E1 -3594.823,E2 -3594.823} C_VEL
LIN {X 0,Y 545.184,Z 135.574,A -85,B 0,C 180,E1 -3597.784,E2 -3597.784} C_VEL
LIN {X 0,Y 545.184,Z 135.578,A -85,B 0,C 180,E1 -3600,E2 -3600} C_VEL
LIN {X 0,Y 545.135,Z 135.575,A -85,B 0,C 180,E1 -3602.956,E2 -3602.956} C_VEL
LIN {X 0,Y 545.118,Z 135.587,A -85,B 0,C 180,E1 -3605.92,E2 -3605.92} C_VEL
LIN {X 0,Y 545.061,Z 135.584,A -85,B 0,C 180,E1 -3608.901,E2 -3608.901} C_VEL
LIN {X 0,Y 545.058,Z 135.593,A -85,B 0,C 180,E1 -3611.906,E2 -3611.906} C_VEL
LIN {X 0,Y 545.069,Z 135.584,A -85,B 0,C 180,E1 -3614.944,E2 -3614.944} C_VEL
LIN {X 0,Y 545.036,Z 135.591,A -85,B 0,C 180,E1 -3618.028,E2 -3618.028} C_VEL
LIN {X 0,Y 545.023,Z 135.59,A -85,B 0,C 180,E1 -3620.375,E2 -3620.375} C_VEL
LIN {X 0,Y 544.981,Z 135.595,A -85,B 0,C 180,E1 -3622.761,E2 -3622.761} C_VEL
LIN {X 0,Y 545.029,Z 135.598,A -85,B 0,C 180,E1 -3625.496,E2 -3625.496} C_VEL
LIN {X 0,Y 545.026,Z 135.589,A -85,B 0,C 180,E1 -3628.497,E2 -3628.497} C_VEL
LIN {X 0,Y 545.039,Z 135.592,A -85,B 0,C 180,E1 -3631.677,E2 -3631.677} C_VEL
LIN {X 0,Y 545.039,Z 135.588,A -85,B 0,C 180,E1 -3634.566,E2 -3634.566} C_VEL
LIN {X 0,Y 545.014,Z 135.599,A -85,B 0,C 180,E1 -3637.306,E2 -3637.306} C_VEL
LIN {X 0,Y 545.029,Z 135.588,A -85,B 0,C 180,E1 -3640.146,E2 -3640.146} C_VEL
LIN {X 0,Y 545.013,Z 135.6,A -85,B 0,C 180,E1 -3643.113,E2 -3643.113} C_VEL
LIN {X 0,Y 545.022,Z 135.59,A -85,B 0,C 180,E1 -3646.23,E2 -3646.23} C_VEL
LIN {X 0,Y 545.012,Z 135.599,A -85,B 0,C 180,E1 -3648.88,E2 -3648.88} C_VEL
LIN {X 0,Y 545.038,Z 135.587,A -85,B 0,C 180,E1 -3651.866,E2 -3651.866} C_VEL
LIN {X 0,Y 545.017,Z 135.595,A -85,B 0,C 180,E1 -3654.531,E2 -3654.531} C_VEL
LIN {X 0,Y 545.049,Z 135.589,A -85,B 0,C 180,E1 -3657.211,E2 -3657.211} C_VEL
LIN {X 0,Y 545.016,Z 135.59,A -85,B 0,C 180,E1 -3659.808,E2 -3659.808} C_VEL
LIN {X 0,Y 544.996,Z 135.598,A -85,B 0,C 180,E1 -3662.339,E2 -3662.339} C_VEL
LIN {X 0,Y 545.021,Z 135.596,A -85,B 0,C 180,E1 -3664.816,E2 -3664.816} C_VEL
LIN {X 0,Y 545.037,Z 135.638,A -85,B 0,C 180,E1 -3666.365,E2 -3666.365} C_VEL
LIN {X 0,Y 546.103,Z 142.354,A -85,B 0,C 180,E1 -3667.472,E2 -3667.472} C_VEL
LIN {X 0,Y 545.892,Z 158.067,A -85,B 0,C 180,E1 -3669.909,E2 -3669.909} C_VEL
LIN {X 0,Y 545.546,Z 176.781,A -85,B 0,C 180,E1 -3672.765,E2 -3672.765} C_VEL
LIN {X 0,Y 545.326,Z 194.521,A -85,B 0,C 180,E1 -3675.445,E2 -3675.445} C_VEL
LIN {X 0,Y 546.483,Z 203.276,A -85,B 0,C 180,E1 -3675.597,E2 -3675.597} C_VEL
LIN {X 0,Y 546.204,Z 302.108,A -85,B 0,C 180,E1 -3676.916,E2 -3676.916} C_VEL
LIN {X 0,Y 546.028,Z 315.569,A -85,B 0,C 180,E1 -3677.243,E2 -3677.243} C_VEL
LIN {X 0,Y 545.856,Z 327.824,A -85,B 0,C 180,E1 -3677.687,E2 -3677.687} C_VEL
LIN {X 0,Y 545.664,Z 339.563,A -85,B 0,C 180,E1 -3678.261,E2 -3678.261} C_VEL
LIN {X 0,Y 545.492,Z 350.519,A -85,B 0,C 180,E1 -3678.951,E2 -3678.951} C_VEL
LIN {X 0,Y 545.249,Z 361.215,A -85,B 0,C 180,E1 -3679.792,E2 -3679.792} C_VEL
LIN {X 0,Y 545.088,Z 370.851,A -85,B 0,C 180,E1 -3680.725,E2 -3680.725} C_VEL
LIN {X 0,Y 544.947,Z 378.747,A -85,B 0,C 180,E1 -3681.658,E2 -3681.658} C_VEL
LIN {X 0,Y 544.824,Z 386.456,A -85,B 0,C 180,E1 -3682.775,E2 -3682.775} C_VEL
LIN {X 0,Y 544.777,Z 393.559,A -85,B 0,C 180,E1 -3684.076,E2 -3684.076} C_VEL
LIN {X 0,Y 544.629,Z 398.279,A -85,B 0,C 180,E1 -3685.188,E2 -3685.188} C_VEL
LIN {X 0,Y 544.669,Z 401.889,A -85,B 0,C 180,E1 -3686.301,E2 -3686.301} C_VEL
LIN {X 0,Y 544.65,Z 403.749,A -85,B 0,C 180,E1 -3687.041,E2 -3687.041} C_VEL
LIN {X 0,Y 544.546,Z 406.137,A -85,B 0,C 180,E1 -3688.521,E2 -3688.521} C_VEL
LIN {X 0,Y 544.542,Z 406.744,A -85,B 0,C 180,E1 -3689.26,E2 -3689.26} C_VEL
LIN {X 0,Y 544.541,Z 406.96,A -85,B 0,C 180,E1 -3690,E2 -3690} C_VEL
LIN {X 0,Y 544.546,Z 406.138,A -85,B 0,C 180,E1 -3691.479,E2 -3691.479} C_VEL
LIN {X 0,Y 544.65,Z 403.752,A -85,B 0,C 180,E1 -3692.958,E2 -3692.958} C_VEL
LIN {X 0,Y 544.684,Z 400.818,A -85,B 0,C 180,E1 -3694.069,E2 -3694.069} C_VEL
LIN {X 0,Y 544.653,Z 396.843,A -85,B 0,C 180,E1 -3695.182,E2 -3695.182} C_VEL
LIN {X 0,Y 544.71,Z 391.572,A -85,B 0,C 180,E1 -3696.326,E2 -3696.326} C_VEL
LIN {X 0,Y 544.836,Z 385.283,A -85,B 0,C 180,E1 -3697.411,E2 -3697.411} C_VEL
LIN {X 0,Y 544.988,Z 377.242,A -85,B 0,C 180,E1 -3698.528,E2 -3698.528} C_VEL
LIN {X 0,Y 545.114,Z 369.042,A -85,B 0,C 180,E1 -3699.461,E2 -3699.461} C_VEL
LIN {X 0,Y 545.353,Z 359.04,A -85,B 0,C 180,E1 -3700.394,E2 -3700.394} C_VEL
LIN {X 0,Y 545.548,Z 348.153,A -85,B 0,C 180,E1 -3701.208,E2 -3701.208} C_VEL
LIN {X 0,Y 545.709,Z 336.649,A -85,B 0,C 180,E1 -3701.891,E2 -3701.891} C_VEL
LIN {X 0,Y 545.927,Z 324.355,A -85,B 0,C 180,E1 -3702.452,E2 -3702.452} C_VEL
LIN {X 0,Y 546.105,Z 311.374,A -85,B 0,C 180,E1 -3702.873,E2 -3702.873} C_VEL
LIN {X 0,Y 546.245,Z 297.533,A -85,B 0,C 180,E1 -3703.154,E2 -3703.154} C_VEL
LIN {X 0,Y 546.409,Z 201.835,A -85,B 0,C 180,E1 -3704.423,E2 -3704.423} C_VEL
LIN {X 0,Y 545.314,Z 194.22,A -85,B 0,C 180,E1 -3704.579,E2 -3704.579} C_VEL
LIN {X 0,Y 545.543,Z 174.217,A -85,B 0,C 180,E1 -3707.576,E2 -3707.576} C_VEL
LIN {X 0,Y 545.916,Z 154.73,A -85,B 0,C 180,E1 -3710.536,E2 -3710.536} C_VEL
LIN {X 0,Y 546.039,Z 141.764,A -85,B 0,C 180,E1 -3712.526,E2 -3712.526} C_VEL
LIN {X 0,Y 545.045,Z 135.596,A -85,B 0,C 180,E1 -3713.56,E2 -3713.56} C_VEL
LIN {X 0,Y 545.039,Z 135.592,A -85,B 0,C 180,E1 -3716.827,E2 -3716.827} C_VEL
LIN {X 0,Y 545.009,Z 135.603,A -85,B 0,C 180,E1 -3719.341,E2 -3719.341} C_VEL
LIN {X 0,Y 545.038,Z 135.591,A -85,B 0,C 180,E1 -3721.915,E2 -3721.915} C_VEL
LIN {X 0,Y 545.04,Z 135.589,A -85,B 0,C 180,E1 -3724.565,E2 -3724.565} C_VEL
LIN {X 0,Y 545.009,Z 135.599,A -85,B 0,C 180,E1 -3727.305,E2 -3727.305} C_VEL
LIN {X 0,Y 545.029,Z 135.59,A -85,B 0,C 180,E1 -3730.145,E2 -3730.145} C_VEL
LIN {X 0,Y 545.012,Z 135.6,A -85,B 0,C 180,E1 -3733.112,E2 -3733.112} C_VEL
LIN {X 0,Y 545.02,Z 135.591,A -85,B 0,C 180,E1 -3736.228,E2 -3736.228} C_VEL
LIN {X 0,Y 545,Z 135.602,A -85,B 0,C 180,E1 -3738.878,E2 -3738.878} C_VEL
LIN {X 0,Y 545.037,Z 135.588,A -85,B 0,C 180,E1 -3741.761,E2 -3741.761} C_VEL
LIN {X 0,Y 545.014,Z 135.596,A -85,B 0,C 180,E1 -3744.53,E2 -3744.53} C_VEL
LIN {X 0,Y 545.054,Z 135.588,A -85,B 0,C 180,E1 -3747.21,E2 -3747.21} C_VEL
LIN {X 0,Y 545.011,Z 135.59,A -85,B 0,C 180,E1 -3749.807,E2 -3749.807} C_VEL
LIN {X 0,Y 545.016,Z 135.594,A -85,B 0,C 180,E1 -3752.841,E2 -3752.841} C_VEL
LIN {X 0,Y 545.009,Z 135.592,A -85,B 0,C 180,E1 -3755.629,E2 -3755.629} C_VEL
LIN {X 0,Y 545.01,Z 135.595,A -85,B 0,C 180,E1 -3758.834,E2 -3758.834} C_VEL
LIN {X 0,Y 545.02,Z 135.589,A -85,B 0,C 180,E1 -3761.193,E2 -3761.193} C_VEL
LIN {X 0,Y 545.013,Z 135.591,A -85,B 0,C 180,E1 -3763.519,E2 -3763.519} C_VEL
LIN {X 0,Y 545.054,Z 135.588,A -85,B 0,C 180,E1 -3765.819,E2 -3765.819} C_VEL
LIN {X 0,Y 545.063,Z 135.585,A -85,B 0,C 180,E1 -3768.848,E2 -3768.848} C_VEL
LIN {X 0,Y 545.057,Z 135.59,A -85,B 0,C 180,E1 -3771.846,E2 -3771.846} C_VEL
LIN {X 0,Y 545.152,Z 135.573,A -85,B 0,C 180,E1 -3774.822,E2 -3774.822} C_VEL
LIN {X 0,Y 545.183,Z 135.576,A -85,B 0,C 180,E1 -3777.783,E2 -3777.783} C_VEL
LIN {X 0,Y 545.182,Z 135.578,A -85,B 0,C 180,E1 -3780,E2 -3780} C_VEL
LIN {X 0,Y 545.133,Z 135.576,A -85,B 0,C 180,E1 -3782.956,E2 -3782.956} C_VEL
LIN {X 0,Y 545.117,Z 135.586,A -85,B 0,C 180,E1 -3785.92,E2 -3785.92} C_VEL
LIN {X 0,Y 545.058,Z 135.586,A -85,B 0,C 180,E1 -3788.901,E2 -3788.901} C_VEL
LIN {X 0,Y 545.056,Z 135.594,A -85,B 0,C 180,E1 -3791.906,E2 -3791.906} C_VEL
LIN {X 0,Y 545.066,Z 135.588,A -85,B 0,C 180,E1 -3794.944,E2 -3794.944} C_VEL
LIN {X 0,Y 545.034,Z 135.592,A -85,B 0,C 180,E1 -3798.027,E2 -3798.027} C_VEL
LIN {X 0,Y 545.038,Z 135.59,A -85,B 0,C 180,E1 -3800.374,E2 -3800.374} C_VEL
LIN {X 0,Y 545.056,Z 135.595,A -85,B 0,C 180,E1 -3803.56,E2 -3803.56} C_VEL
LIN {X 0,Y 545.091,Z 135.793,A -85,B 0,C 180,E1 -3804.048,E2 -3804.048} C_VEL
LIN {X 0,Y 545.487,Z 140.898,A -85,B 0,C 180,E1 -3804.957,E2 -3804.957} C_VEL
LIN {X 0,Y 545.344,Z 156.165,A -85,B 0,C 180,E1 -3807.641,E2 -3807.641} C_VEL
LIN {X 0,Y 545.24,Z 166.487,A -85,B 0,C 180,E1 -3809.487,E2 -3809.487} C_VEL
LIN {X 0,Y 546.57,Z 175.45,A -85,B 0,C 180,E1 -3809.659,E2 -3809.659} C_VEL
LIN {X 0,Y 546.405,Z 218.998,A -85,B 0,C 180,E1 -3810.238,E2 -3810.238} C_VEL
LIN {X 0,Y 545.737,Z 224.844,A -85,B 0,C 180,E1 -3810.298,E2 -3810.298} C_VEL
LIN {X 0,Y 540.022,Z 243.828,A -85,B 0,C 180,E1 -3810.405,E2 -3810.405} C_VEL
LIN {X 0,Y 539.412,Z 249.669,A -85,B 0,C 180,E1 -3810.468,E2 -3810.468} C_VEL
LIN {X 0,Y 539.238,Z 275.312,A -85,B 0,C 180,E1 -3810.841,E2 -3810.841} C_VEL
LIN {X 0,Y 539.115,Z 287.813,A -85,B 0,C 180,E1 -3811.171,E2 -3811.171} C_VEL
LIN {X 0,Y 538.956,Z 300.957,A -85,B 0,C 180,E1 -3811.676,E2 -3811.676} C_VEL
LIN {X 0,Y 538.657,Z 313.458,A -85,B 0,C 180,E1 -3812.339,E2 -3812.339} C_VEL
LIN {X 0,Y 538.455,Z 323.507,A -85,B 0,C 180,E1 -3813.019,E2 -3813.019} C_VEL
LIN {X 0,Y 538.26,Z 333.238,A -85,B 0,C 180,E1 -3813.826,E2 -3813.826} C_VEL
LIN {X 0,Y 538.052,Z 343.088,A -85,B 0,C 180,E1 -3814.825,E2 -3814.825} C_VEL
LIN {X 0,Y 537.847,Z 352.359,A -85,B 0,C 180,E1 -3816.016,E2 -3816.016} C_VEL
LIN {X 0,Y 537.712,Z 359.316,A -85,B 0,C 180,E1 -3817.13,E2 -3817.13} C_VEL
LIN {X 0,Y 537.667,Z 364.372,A -85,B 0,C 180,E1 -3818.125,E2 -3818.125} C_VEL
LIN {X 0,Y 537.594,Z 368.754,A -85,B 0,C 180,E1 -3819.195,E2 -3819.195} C_VEL
LIN {X 0,Y 537.546,Z 372.135,A -85,B 0,C 180,E1 -3820.258,E2 -3820.258} C_VEL
LIN {X 0,Y 537.512,Z 373.635,A -85,B 0,C 180,E1 -3820.825,E2 -3820.825} C_VEL
LIN {X 0,Y 537.493,Z 375.573,A -85,B 0,C 180,E1 -3821.824,E2 -3821.824} C_VEL
LIN {X 0,Y 537.488,Z 376.872,A -85,B 0,C 180,E1 -3822.927,E2 -3822.927} C_VEL
LIN {X 0,Y 537.493,Z 377.309,A -85,B 0,C 180,E1 -3824.016,E2 -3824.016} C_VEL
LIN {X 0,Y 537.519,Z 376.917,A -85,B 0,C 180,E1 -3825.087,E2 -3825.087} C_VEL
LIN {X 0,Y 537.474,Z 375.764,A -85,B 0,C 180,E1 -3826.131,E2 -3826.131} C_VEL
LIN {X 0,Y 537.522,Z 373.828,A -85,B 0,C 180,E1 -3827.166,E2 -3827.166} C_VEL
LIN {X 0,Y 537.568,Z 369.518,A -85,B 0,C 180,E1 -3828.684,E2 -3828.684} C_VEL
LIN {X 0,Y 537.627,Z 364.401,A -85,B 0,C 180,E1 -3829.955,E2 -3829.955} C_VEL
LIN {X 0,Y 537.729,Z 360.175,A -85,B 0,C 180,E1 -3830.802,E2 -3830.802} C_VEL
LIN {X 0,Y 537.814,Z 353.696,A -85,B 0,C 180,E1 -3831.872,E2 -3831.872} C_VEL
LIN {X 0,Y 537.958,Z 346.599,A -85,B 0,C 180,E1 -3832.836,E2 -3832.836} C_VEL
LIN {X 0,Y 538.154,Z 338.25,A -85,B 0,C 180,E1 -3833.777,E2 -3833.777} C_VEL
LIN {X 0,Y 538.353,Z 328.099,A -85,B 0,C 180,E1 -3834.714,E2 -3834.714} C_VEL
LIN {X 0,Y 538.579,Z 317.834,A -85,B 0,C 180,E1 -3835.473,E2 -3835.473} C_VEL
LIN {X 0,Y 538.804,Z 307.824,A -85,B 0,C 180,E1 -3836.07,E2 -3836.07} C_VEL
LIN {X 0,Y 538.974,Z 297.362,A -85,B 0,C 180,E1 -3836.567,E2 -3836.567} C_VEL
LIN {X 0,Y 539.166,Z 285.506,A -85,B 0,C 180,E1 -3836.988,E2 -3836.988} C_VEL
LIN {X 0,Y 539.297,Z 273.274,A -85,B 0,C 180,E1 -3837.289,E2 -3837.289} C_VEL
LIN {X 0,Y 539.666,Z 174.82,A -85,B 0,C 180,E1 -3838.634,E2 -3838.634} C_VEL
LIN {X 0,Y 538.262,Z 166.731,A -85,B 0,C 180,E1 -3838.79,E2 -3838.79} C_VEL
LIN {X 0,Y 538.525,Z 149.366,A -85,B 0,C 180,E1 -3841.978,E2 -3841.978} C_VEL
LIN {X 0,Y 538.65,Z 140.237,A -85,B 0,C 180,E1 -3843.666,E2 -3843.666} C_VEL
LIN {X 0,Y 538.037,Z 136.469,A -85,B 0,C 180,E1 -3844.412,E2 -3844.412} C_VEL
LIN {X 0,Y 537.97,Z 136.474,A -85,B 0,C 180,E1 -3846.927,E2 -3846.927} C_VEL
LIN {X 0,Y 538.053,Z 136.462,A -85,B 0,C 180,E1 -3850.127,E2 -3850.127} C_VEL
LIN {X 0,Y 537.964,Z 136.469,A -85,B 0,C 180,E1 -3853.297,E2 -3853.297} C_VEL
LIN {X 0,Y 538.036,Z 136.46,A -85,B 0,C 180,E1 -3855.63,E2 -3855.63} C_VEL
LIN {X 0,Y 538.019,Z 136.466,A -85,B 0,C 180,E1 -3858.701,E2 -3858.701} C_VEL
LIN {X 0,Y 538.03,Z 136.462,A -85,B 0,C 180,E1 -3861.739,E2 -3861.739} C_VEL
LIN {X 0,Y 538.117,Z 136.452,A -85,B 0,C 180,E1 -3864.755,E2 -3864.755} C_VEL
LIN {X 0,Y 538.158,Z 136.448,A -85,B 0,C 180,E1 -3867.755,E2 -3867.755} C_VEL
LIN {X 0,Y 538.156,Z 136.453,A -85,B 0,C 180,E1 -3870,E2 -3870} C_VEL
LIN {X 0,Y 538.106,Z 136.451,A -85,B 0,C 180,E1 -3872.995,E2 -3872.995} C_VEL
LIN {X 0,Y 538.076,Z 136.464,A -85,B 0,C 180,E1 -3875.998,E2 -3875.998} C_VEL
LIN {X 0,Y 538.021,Z 136.462,A -85,B 0,C 180,E1 -3879.018,E2 -3879.018} C_VEL
LIN {X 0,Y 538.031,Z 136.466,A -85,B 0,C 180,E1 -3882.064,E2 -3882.064} C_VEL
LIN {X 0,Y 538.032,Z 136.462,A -85,B 0,C 180,E1 -3885.144,E2 -3885.144} C_VEL
LIN {X 0,Y 537.991,Z 136.467,A -85,B 0,C 180,E1 -3888.271,E2 -3888.271} C_VEL
LIN {X 0,Y 537.982,Z 136.466,A -85,B 0,C 180,E1 -3890.653,E2 -3890.653} C_VEL
LIN {X 0,Y 537.971,Z 136.47,A -85,B 0,C 180,E1 -3893.074,E2 -3893.074} C_VEL
LIN {X 0,Y 537.989,Z 136.473,A -85,B 0,C 180,E1 -3895.661,E2 -3895.661} C_VEL
LIN {X 0,Y 537.966,Z 136.47,A -85,B 0,C 180,E1 -3898.054,E2 -3898.054} C_VEL
LIN {X 0,Y 537.987,Z 136.466,A -85,B 0,C 180,E1 -3900.629,E2 -3900.629} C_VEL
LIN {X 0,Y 538.015,Z 136.471,A -85,B 0,C 180,E1 -3903.278,E2 -3903.278} C_VEL
LIN {X 0,Y 537.963,Z 136.469,A -85,B 0,C 180,E1 -3906.007,E2 -3906.007} C_VEL
LIN {X 0,Y 538,Z 136.468,A -85,B 0,C 180,E1 -3908.831,E2 -3908.831} C_VEL
LIN {X 0,Y 537.973,Z 136.468,A -85,B 0,C 180,E1 -3911.872,E2 -3911.872} C_VEL
LIN {X 0,Y 537.987,Z 136.472,A -85,B 0,C 180,E1 -3914.864,E2 -3914.864} C_VEL
LIN {X 0,Y 537.965,Z 136.475,A -85,B 0,C 180,E1 -3917.209,E2 -3917.209} C_VEL
LIN {X 0,Y 537.997,Z 136.465,A -85,B 0,C 180,E1 -3920.201,E2 -3920.201} C_VEL
LIN {X 0,Y 537.965,Z 136.475,A -85,B 0,C 180,E1 -3923.063,E2 -3923.063} C_VEL
LIN {X 0,Y 537.989,Z 136.465,A -85,B 0,C 180,E1 -3925.825,E2 -3925.825} C_VEL
LIN {X 0,Y 537.986,Z 136.471,A -85,B 0,C 180,E1 -3928.498,E2 -3928.498} C_VEL
LIN {X 0,Y 537.977,Z 136.471,A -85,B 0,C 180,E1 -3931.095,E2 -3931.095} C_VEL
LIN {X 0,Y 537.976,Z 136.467,A -85,B 0,C 180,E1 -3933.63,E2 -3933.63} C_VEL
LIN {X 0,Y 537.976,Z 136.47,A -85,B 0,C 180,E1 -3936.128,E2 -3936.128} C_VEL
LIN {X 0,Y 537.99,Z 136.475,A -85,B 0,C 180,E1 -3938.545,E2 -3938.545} C_VEL
LIN {X 0,Y 537.997,Z 136.467,A -85,B 0,C 180,E1 -3940.939,E2 -3940.939} C_VEL
LIN {X 0,Y 537.961,Z 136.469,A -85,B 0,C 180,E1 -3943.297,E2 -3943.297} C_VEL
LIN {X 0,Y 538.033,Z 136.461,A -85,B 0,C 180,E1 -3945.63,E2 -3945.63} C_VEL
LIN {X 0,Y 538.016,Z 136.466,A -85,B 0,C 180,E1 -3948.701,E2 -3948.701} C_VEL
LIN {X 0,Y 538.027,Z 136.463,A -85,B 0,C 180,E1 -3951.739,E2 -3951.739} C_VEL
LIN {X 0,Y 538.114,Z 136.452,A -85,B 0,C 180,E1 -3954.755,E2 -3954.755} C_VEL
LIN {X 0,Y 538.155,Z 136.449,A -85,B 0,C 180,E1 -3957.755,E2 -3957.755} C_VEL
LIN {X 0,Y 538.152,Z 136.454,A -85,B 0,C 180,E1 -3960,E2 -3960} C_VEL
LIN {X 0,Y 538.103,Z 136.451,A -85,B 0,C 180,E1 -3962.995,E2 -3962.995} C_VEL
LIN {X 0,Y 538.074,Z 136.463,A -85,B 0,C 180,E1 -3965.998,E2 -3965.998} C_VEL
LIN {X 0,Y 538.019,Z 136.462,A -85,B 0,C 180,E1 -3969.019,E2 -3969.019} C_VEL
LIN {X 0,Y 538.029,Z 136.466,A -85,B 0,C 180,E1 -3972.064,E2 -3972.064} C_VEL
LIN {X 0,Y 538.03,Z 136.462,A -85,B 0,C 180,E1 -3975.145,E2 -3975.145} C_VEL
LIN {X 0,Y 537.989,Z 136.467,A -85,B 0,C 180,E1 -3978.272,E2 -3978.272} C_VEL
LIN {X 0,Y 537.981,Z 136.466,A -85,B 0,C 180,E1 -3980.654,E2 -3980.654} C_VEL
LIN {X 0,Y 537.969,Z 136.471,A -85,B 0,C 180,E1 -3983.074,E2 -3983.074} C_VEL
LIN {X 0,Y 537.988,Z 136.472,A -85,B 0,C 180,E1 -3985.661,E2 -3985.661} C_VEL
LIN {X 0,Y 537.966,Z 136.47,A -85,B 0,C 180,E1 -3988.054,E2 -3988.054} C_VEL
LIN {X 0,Y 537.983,Z 136.467,A -85,B 0,C 180,E1 -3990.63,E2 -3990.63} C_VEL
LIN {X 0,Y 538.016,Z 136.471,A -85,B 0,C 180,E1 -3993.279,E2 -3993.279} C_VEL
LIN {X 0,Y 537.956,Z 136.47,A -85,B 0,C 180,E1 -3996.008,E2 -3996.008} C_VEL
LIN {X 0,Y 537.996,Z 136.469,A -85,B 0,C 180,E1 -3998.832,E2 -3998.832} C_VEL
LIN {X 0,Y 537.973,Z 136.468,A -85,B 0,C 180,E1 -4001.873,E2 -4001.873} C_VEL
LIN {X 0,Y 537.99,Z 136.472,A -85,B 0,C 180,E1 -4004.864,E2 -4004.864} C_VEL
LIN {X 0,Y 537.968,Z 136.474,A -85,B 0,C 180,E1 -4007.21,E2 -4007.21} C_VEL
LIN {X 0,Y 537.985,Z 136.467,A -85,B 0,C 180,E1 -4010.2,E2 -4010.2} C_VEL
LIN {X 0,Y 537.957,Z 136.476,A -85,B 0,C 180,E1 -4013.062,E2 -4013.062} C_VEL
LIN {X 0,Y 537.993,Z 136.465,A -85,B 0,C 180,E1 -4015.825,E2 -4015.825} C_VEL
LIN {X 0,Y 537.988,Z 136.471,A -85,B 0,C 180,E1 -4018.498,E2 -4018.498} C_VEL
LIN {X 0,Y 537.984,Z 136.47,A -85,B 0,C 180,E1 -4021.096,E2 -4021.096} C_VEL
LIN {X 0,Y 537.976,Z 136.467,A -85,B 0,C 180,E1 -4023.63,E2 -4023.63} C_VEL
LIN {X 0,Y 538.002,Z 136.585,A -85,B 0,C 180,E1 -4026.213,E2 -4026.213} C_VEL
LIN {X 0,Y 539.183,Z 143.839,A -85,B 0,C 180,E1 -4027.427,E2 -4027.427} C_VEL
LIN {X 0,Y 538.896,Z 159.468,A -85,B 0,C 180,E1 -4029.883,E2 -4029.883} C_VEL
LIN {X 0,Y 538.544,Z 176.612,A -85,B 0,C 180,E1 -4032.534,E2 -4032.534} C_VEL
LIN {X 0,Y 538.298,Z 194.511,A -85,B 0,C 180,E1 -4035.255,E2 -4035.255} C_VEL
LIN {X 0,Y 539.596,Z 203.428,A -85,B 0,C 180,E1 -4035.414,E2 -4035.414} C_VEL
LIN {X 0,Y 539.272,Z 302.871,A -85,B 0,C 180,E1 -4036.769,E2 -4036.769} C_VEL
LIN {X 0,Y 539.088,Z 315.993,A -85,B 0,C 180,E1 -4037.1,E2 -4037.1} C_VEL
LIN {X 0,Y 538.89,Z 328.651,A -85,B 0,C 180,E1 -4037.574,E2 -4037.574} C_VEL
LIN {X 0,Y 538.657,Z 340.245,A -85,B 0,C 180,E1 -4038.162,E2 -4038.162} C_VEL
LIN {X 0,Y 538.466,Z 351.562,A -85,B 0,C 180,E1 -4038.9,E2 -4038.9} C_VEL
LIN {X 0,Y 538.2,Z 362.046,A -85,B 0,C 180,E1 -4039.751,E2 -4039.751} C_VEL
LIN {X 0,Y 538.048,Z 370.619,A -85,B 0,C 180,E1 -4040.603,E2 -4040.603} C_VEL
LIN {X 0,Y 537.899,Z 378.525,A -85,B 0,C 180,E1 -4041.548,E2 -4041.548} C_VEL
LIN {X 0,Y 537.755,Z 386.243,A -85,B 0,C 180,E1 -4042.679,E2 -4042.679} C_VEL
LIN {X 0,Y 537.685,Z 393.351,A -85,B 0,C 180,E1 -4043.998,E2 -4043.998} C_VEL
LIN {X 0,Y 537.54,Z 398.077,A -85,B 0,C 180,E1 -4045.125,E2 -4045.125} C_VEL
LIN {X 0,Y 537.591,Z 401.691,A -85,B 0,C 180,E1 -4046.252,E2 -4046.252} C_VEL
LIN {X 0,Y 537.551,Z 403.553,A -85,B 0,C 180,E1 -4047.002,E2 -4047.002} C_VEL
LIN {X 0,Y 537.451,Z 405.942,A -85,B 0,C 180,E1 -4048.501,E2 -4048.501} C_VEL
LIN {X 0,Y 537.444,Z 406.55,A -85,B 0,C 180,E1 -4049.251,E2 -4049.251} C_VEL
LIN {X 0,Y 537.445,Z 406.766,A -85,B 0,C 180,E1 -4050,E2 -4050} C_VEL
LIN {X 0,Y 537.451,Z 405.942,A -85,B 0,C 180,E1 -4051.498,E2 -4051.498} C_VEL
LIN {X 0,Y 537.49,Z 404.947,A -85,B 0,C 180,E1 -4052.248,E2 -4052.248} C_VEL
LIN {X 0,Y 537.551,Z 403.55,A -85,B 0,C 180,E1 -4052.998,E2 -4052.998} C_VEL
LIN {X 0,Y 537.603,Z 400.612,A -85,B 0,C 180,E1 -4054.123,E2 -4054.123} C_VEL
LIN {X 0,Y 537.587,Z 396.631,A -85,B 0,C 180,E1 -4055.25,E2 -4055.25} C_VEL
LIN {X 0,Y 537.616,Z 391.857,A -85,B 0,C 180,E1 -4056.308,E2 -4056.308} C_VEL
LIN {X 0,Y 537.754,Z 385.052,A -85,B 0,C 180,E1 -4057.509,E2 -4057.509} C_VEL
LIN {X 0,Y 537.912,Z 377.001,A -85,B 0,C 180,E1 -4058.641,E2 -4058.641} C_VEL
LIN {X 0,Y 538.07,Z 368.79,A -85,B 0,C 180,E1 -4059.586,E2 -4059.586} C_VEL
LIN {X 0,Y 538.326,Z 358.772,A -85,B 0,C 180,E1 -4060.531,E2 -4060.531} C_VEL
LIN {X 0,Y 538.541,Z 348.874,A -85,B 0,C 180,E1 -4061.288,E2 -4061.288} C_VEL
LIN {X 0,Y 538.711,Z 337.846,A -85,B 0,C 180,E1 -4061.967,E2 -4061.967} C_VEL
LIN {X 0,Y 538.96,Z 325.149,A -85,B 0,C 180,E1 -4062.568,E2 -4062.568} C_VEL
LIN {X 0,Y 539.139,Z 312.774,A -85,B 0,C 180,E1 -4062.995,E2 -4062.995} C_VEL
LIN {X 0,Y 539.317,Z 299.996,A -85,B 0,C 180,E1 -4063.278,E2 -4063.278} C_VEL
LIN {X 0,Y 539.447,Z 202.019,A -85,B 0,C 180,E1 -4064.608,E2 -4064.608} C_VEL
LIN {X 0,Y 538.246,Z 194.079,A -85,B 0,C 180,E1 -4064.763,E2 -4064.763} C_VEL
LIN {X 0,Y 538.52,Z 176.25,A -85,B 0,C 180,E1 -4067.467,E2 -4067.467} C_VEL
LIN {X 0,Y 538.872,Z 157.79,A -85,B 0,C 180,E1 -4070.301,E2 -4070.301} C_VEL
LIN {X 0,Y 539.08,Z 142.882,A -85,B 0,C 180,E1 -4072.618,E2 -4072.618} C_VEL
LIN {X 0,Y 537.992,Z 136.474,A -85,B 0,C 180,E1 -4073.675,E2 -4073.675} C_VEL
LIN {X 0,Y 537.975,Z 136.47,A -85,B 0,C 180,E1 -4076.37,E2 -4076.37} C_VEL
LIN {X 0,Y 537.972,Z 136.474,A -85,B 0,C 180,E1 -4078.921,E2 -4078.921} C_VEL
LIN {X 0,Y 537.993,Z 136.469,A -85,B 0,C 180,E1 -4081.884,E2 -4081.884} C_VEL
LIN {X 0,Y 537.991,Z 136.468,A -85,B 0,C 180,E1 -4084.614,E2 -4084.614} C_VEL
LIN {X 0,Y 537.977,Z 136.469,A -85,B 0,C 180,E1 -4087.878,E2 -4087.878} C_VEL
LIN {X 0,Y 537.986,Z 136.473,A -85,B 0,C 180,E1 -4090.781,E2 -4090.781} C_VEL
LIN {X 0,Y 537.996,Z 136.466,A -85,B 0,C 180,E1 -4094.07,E2 -4094.07} C_VEL
LIN {X 0,Y 537.964,Z 136.476,A -85,B 0,C 180,E1 -4097.019,E2 -4097.019} C_VEL
LIN {X 0,Y 537.985,Z 136.47,A -85,B 0,C 180,E1 -4099.26,E2 -4099.26} C_VEL
LIN {X 0,Y 537.976,Z 136.469,A -85,B 0,C 180,E1 -4102.121,E2 -4102.121} C_VEL
LIN {X 0,Y 537.988,Z 136.467,A -85,B 0,C 180,E1 -4105.385,E2 -4105.385} C_VEL
LIN {X 0,Y 537.991,Z 136.467,A -85,B 0,C 180,E1 -4108.115,E2 -4108.115} C_VEL
LIN {X 0,Y 537.978,Z 136.47,A -85,B 0,C 180,E1 -4111.095,E2 -4111.095} C_VEL
LIN {X 0,Y 537.976,Z 136.466,A -85,B 0,C 180,E1 -4113.63,E2 -4113.63} C_VEL
LIN {X 0,Y 537.976,Z 136.472,A -85,B 0,C 180,E1 -4116.127,E2 -4116.127} C_VEL
LIN {X 0,Y 537.982,Z 136.475,A -85,B 0,C 180,E1 -4118.544,E2 -4118.544} C_VEL
LIN {X 0,Y 537.977,Z 136.467,A -85,B 0,C 180,E1 -4120.938,E2 -4120.938} C_VEL
LIN {X 0,Y 537.961,Z 136.469,A -85,B 0,C 180,E1 -4123.297,E2 -4123.297} C_VEL
LIN {X 0,Y 538.028,Z 136.461,A -85,B 0,C 180,E1 -4125.629,E2 -4125.629} C_VEL
LIN {X 0,Y 538.015,Z 136.465,A -85,B 0,C 180,E1 -4128.7,E2 -4128.7} C_VEL
LIN {X 0,Y 538.025,Z 136.464,A -85,B 0,C 180,E1 -4131.738,E2 -4131.738} C_VEL
LIN {X 0,Y 538.112,Z 136.45,A -85,B 0,C 180,E1 -4134.754,E2 -4134.754} C_VEL
LIN {X 0,Y 538.154,Z 136.451,A -85,B 0,C 180,E1 -4137.754,E2 -4137.754} C_VEL
LIN {X 0,Y 538.151,Z 136.454,A -85,B 0,C 180,E1 -4140,E2 -4140} C_VEL
LIN {X 0,Y 538.101,Z 136.452,A -85,B 0,C 180,E1 -4142.994,E2 -4142.994} C_VEL
LIN {X 0,Y 538.072,Z 136.463,A -85,B 0,C 180,E1 -4145.998,E2 -4145.998} C_VEL
LIN {X 0,Y 538.017,Z 136.464,A -85,B 0,C 180,E1 -4149.018,E2 -4149.018} C_VEL
LIN {X 0,Y 538.027,Z 136.467,A -85,B 0,C 180,E1 -4152.063,E2 -4152.063} C_VEL
LIN {X 0,Y 538.026,Z 136.467,A -85,B 0,C 180,E1 -4155.144,E2 -4155.144} C_VEL
LIN {X 0,Y 537.99,Z 136.468,A -85,B 0,C 180,E1 -4158.271,E2 -4158.271} C_VEL
LIN {X 0,Y 537.993,Z 136.468,A -85,B 0,C 180,E1 -4160.653,E2 -4160.653} C_VEL
LIN {X 0,Y 538.048,Z 136.623,A -85,B 0,C 180,E1 -4163.937,E2 -4163.937} C_VEL
LIN {X 0,Y 538.508,Z 140.761,A -85,B 0,C 180,E1 -4164.685,E2 -4164.685} C_VEL
LIN {X 0,Y 538.344,Z 154.888,A -85,B 0,C 180,E1 -4167.188,E2 -4167.188} C_VEL
LIN {X 0,Y 538.254,Z 166.769,A -85,B 0,C 180,E1 -4169.305,E2 -4169.305} C_VEL
LIN {X 0,Y 539.706,Z 175.993,A -85,B 0,C 180,E1 -4169.479,E2 -4169.479} C_VEL
LIN {X 0,Y 539.412,Z 249.669,A -85,B 0,C 180,E1 -4170.468,E2 -4170.468} C_VEL
LIN {X 0,Y 538.825,Z 255.517,A -85,B 0,C 180,E1 -4170.529,E2 -4170.529} C_VEL
LIN {X 0,Y 533.128,Z 274.472,A -85,B 0,C 180,E1 -4170.666,E2 -4170.666} C_VEL
LIN {X 0,Y 532.311,Z 280.227,A -85,B 0,C 180,E1 -4170.779,E2 -4170.779} C_VEL
LIN {X 0,Y 532.109,Z 294.234,A -85,B 0,C 180,E1 -4171.225,E2 -4171.225} C_VEL
LIN {X 0,Y 531.882,Z 305.655,A -85,B 0,C 180,E1 -4171.739,E2 -4171.739} C_VEL
LIN {X 0,Y 531.639,Z 316.99,A -85,B 0,C 180,E1 -4172.399,E2 -4172.399} C_VEL
LIN {X 0,Y 531.386,Z 328.926,A -85,B 0,C 180,E1 -4173.289,E2 -4173.289} C_VEL
LIN {X 0,Y 531.163,Z 338.763,A -85,B 0,C 180,E1 -4174.217,E2 -4174.217} C_VEL
LIN {X 0,Y 530.926,Z 347.38,A -85,B 0,C 180,E1 -4175.209,E2 -4175.209} C_VEL
LIN {X 0,Y 530.77,Z 355.275,A -85,B 0,C 180,E1 -4176.321,E2 -4176.321} C_VEL
LIN {X 0,Y 530.628,Z 362.187,A -85,B 0,C 180,E1 -4177.535,E2 -4177.535} C_VEL
LIN {X 0,Y 530.546,Z 366.987,A -85,B 0,C 180,E1 -4178.598,E2 -4178.598} C_VEL
LIN {X 0,Y 530.485,Z 371.179,A -85,B 0,C 180,E1 -4179.791,E2 -4179.791} C_VEL
LIN {X 0,Y 530.42,Z 374.186,A -85,B 0,C 180,E1 -4180.955,E2 -4180.955} C_VEL
LIN {X 0,Y 530.376,Z 376.661,A -85,B 0,C 180,E1 -4182.516,E2 -4182.516} C_VEL
LIN {X 0,Y 530.366,Z 377.372,A -85,B 0,C 180,E1 -4183.556,E2 -4183.556} C_VEL
LIN {X 0,Y 530.404,Z 377.338,A -85,B 0,C 180,E1 -4184.608,E2 -4184.608} C_VEL
LIN {X 0,Y 530.401,Z 376.521,A -85,B 0,C 180,E1 -4185.685,E2 -4185.685} C_VEL
LIN {X 0,Y 530.404,Z 374.856,A -85,B 0,C 180,E1 -4186.782,E2 -4186.782} C_VEL
LIN {X 0,Y 530.451,Z 372.276,A -85,B 0,C 180,E1 -4187.897,E2 -4187.897} C_VEL
LIN {X 0,Y 530.521,Z 368.665,A -85,B 0,C 180,E1 -4189.033,E2 -4189.033} C_VEL
LIN {X 0,Y 530.6,Z 363.854,A -85,B 0,C 180,E1 -4190.195,E2 -4190.195} C_VEL
LIN {X 0,Y 530.73,Z 356.868,A -85,B 0,C 180,E1 -4191.511,E2 -4191.511} C_VEL
LIN {X 0,Y 530.866,Z 349.605,A -85,B 0,C 180,E1 -4192.591,E2 -4192.591} C_VEL
LIN {X 0,Y 531.072,Z 341.649,A -85,B 0,C 180,E1 -4193.559,E2 -4193.559} C_VEL
LIN {X 0,Y 531.311,Z 332.256,A -85,B 0,C 180,E1 -4194.499,E2 -4194.499} C_VEL
LIN {X 0,Y 531.531,Z 323.176,A -85,B 0,C 180,E1 -4195.249,E2 -4195.249} C_VEL
LIN {X 0,Y 531.734,Z 312.985,A -85,B 0,C 180,E1 -4195.94,E2 -4195.94} C_VEL
LIN {X 0,Y 531.976,Z 300.926,A -85,B 0,C 180,E1 -4196.583,E2 -4196.583} C_VEL
LIN {X 0,Y 532.194,Z 287.747,A -85,B 0,C 180,E1 -4197.093,E2 -4197.093} C_VEL
LIN {X 0,Y 532.344,Z 274.804,A -85,B 0,C 180,E1 -4197.433,E2 -4197.433} C_VEL
LIN {X 0,Y 532.793,Z 175.465,A -85,B 0,C 180,E1 -4198.82,E2 -4198.82} C_VEL
LIN {X 0,Y 531.295,Z 166.836,A -85,B 0,C 180,E1 -4198.998,E2 -4198.998} C_VEL
LIN {X 0,Y 531.538,Z 150.591,A -85,B 0,C 180,E1 -4202.007,E2 -4202.007} C_VEL
LIN {X 0,Y 531.681,Z 141.453,A -85,B 0,C 180,E1 -4203.717,E2 -4203.717} C_VEL
LIN {X 0,Y 530.992,Z 137.346,A -85,B 0,C 180,E1 -4204.523,E2 -4204.523} C_VEL
LIN {X 0,Y 530.953,Z 137.345,A -85,B 0,C 180,E1 -4207.904,E2 -4207.904} C_VEL
LIN {X 0,Y 530.957,Z 137.349,A -85,B 0,C 180,E1 -4210.676,E2 -4210.676} C_VEL
LIN {X 0,Y 530.932,Z 137.346,A -85,B 0,C 180,E1 -4213.07,E2 -4213.07} C_VEL
LIN {X 0,Y 530.997,Z 137.337,A -85,B 0,C 180,E1 -4215.436,E2 -4215.436} C_VEL
LIN {X 0,Y 530.981,Z 137.345,A -85,B 0,C 180,E1 -4218.549,E2 -4218.549} C_VEL
LIN {X 0,Y 530.978,Z 137.34,A -85,B 0,C 180,E1 -4221.628,E2 -4221.628} C_VEL
LIN {X 0,Y 531.078,Z 137.329,A -85,B 0,C 180,E1 -4224.685,E2 -4224.685} C_VEL
LIN {X 0,Y 531.129,Z 137.323,A -85,B 0,C 180,E1 -4227.725,E2 -4227.725} C_VEL
LIN {X 0,Y 531.124,Z 137.329,A -85,B 0,C 180,E1 -4230,E2 -4230} C_VEL
LIN {X 0,Y 531.13,Z 137.326,A -85,B 0,C 180,E1 -4232.275,E2 -4232.275} C_VEL
LIN {X 0,Y 531.078,Z 137.328,A -85,B 0,C 180,E1 -4235.315,E2 -4235.315} C_VEL
LIN {X 0,Y 530.978,Z 137.341,A -85,B 0,C 180,E1 -4238.372,E2 -4238.372} C_VEL
LIN {X 0,Y 531.007,Z 137.342,A -85,B 0,C 180,E1 -4241.65,E2 -4241.65} C_VEL
LIN {X 0,Y 531.015,Z 137.335,A -85,B 0,C 180,E1 -4244.95,E2 -4244.95} C_VEL
LIN {X 0,Y 530.967,Z 137.349,A -85,B 0,C 180,E1 -4247.724,E2 -4247.724} C_VEL
LIN {X 0,Y 530.967,Z 137.343,A -85,B 0,C 180,E1 -4250.129,E2 -4250.129} C_VEL
LIN {X 0,Y 530.912,Z 137.347,A -85,B 0,C 180,E1 -4252.575,E2 -4252.575} C_VEL
LIN {X 0,Y 530.943,Z 137.346,A -85,B 0,C 180,E1 -4255.06,E2 -4255.06} C_VEL
LIN {X 0,Y 530.945,Z 137.35,A -85,B 0,C 180,E1 -4257.599,E2 -4257.599} C_VEL
LIN {X 0,Y 530.941,Z 137.344,A -85,B 0,C 180,E1 -4260.64,E2 -4260.64} C_VEL
LIN {X 0,Y 530.955,Z 137.348,A -85,B 0,C 180,E1 -4263.499,E2 -4263.499} C_VEL
LIN {X 0,Y 530.937,Z 137.345,A -85,B 0,C 180,E1 -4266.559,E2 -4266.559} C_VEL
LIN {X 0,Y 530.958,Z 137.347,A -85,B 0,C 180,E1 -4269.445,E2 -4269.445} C_VEL
LIN {X 0,Y 530.907,Z 137.349,A -85,B 0,C 180,E1 -4272.463,E2 -4272.463} C_VEL
LIN {X 0,Y 530.957,Z 137.345,A -85,B 0,C 180,E1 -4275.45,E2 -4275.45} C_VEL
LIN {X 0,Y 530.948,Z 137.346,A -85,B 0,C 180,E1 -4278.561,E2 -4278.561} C_VEL
LIN {X 0,Y 530.942,Z 137.345,A -85,B 0,C 180,E1 -4281.528,E2 -4281.528} C_VEL
LIN {X 0,Y 530.923,Z 137.348,A -85,B 0,C 180,E1 -4284.378,E2 -4284.378} C_VEL
LIN {X 0,Y 530.957,Z 137.346,A -85,B 0,C 180,E1 -4287.133,E2 -4287.133} C_VEL
LIN {X 0,Y 530.924,Z 137.346,A -85,B 0,C 180,E1 -4289.801,E2 -4289.801} C_VEL
LIN {X 0,Y 530.947,Z 137.349,A -85,B 0,C 180,E1 -4292.48,E2 -4292.48} C_VEL
LIN {X 0,Y 530.939,Z 137.348,A -85,B 0,C 180,E1 -4294.939,E2 -4294.939} C_VEL
LIN {X 0,Y 530.943,Z 137.348,A -85,B 0,C 180,E1 -4298.246,E2 -4298.246} C_VEL
LIN {X 0,Y 530.954,Z 137.348,A -85,B 0,C 180,E1 -4300.676,E2 -4300.676} C_VEL
LIN {X 0,Y 530.929,Z 137.346,A -85,B 0,C 180,E1 -4303.069,E2 -4303.069} C_VEL
LIN {X 0,Y 530.993,Z 137.337,A -85,B 0,C 180,E1 -4305.435,E2 -4305.435} C_VEL
LIN {X 0,Y 530.978,Z 137.345,A -85,B 0,C 180,E1 -4308.549,E2 -4308.549} C_VEL
LIN {X 0,Y 530.975,Z 137.341,A -85,B 0,C 180,E1 -4311.629,E2 -4311.629} C_VEL
LIN {X 0,Y 531.075,Z 137.329,A -85,B 0,C 180,E1 -4314.685,E2 -4314.685} C_VEL
LIN {X 0,Y 531.127,Z 137.324,A -85,B 0,C 180,E1 -4317.725,E2 -4317.725} C_VEL
LIN {X 0,Y 531.121,Z 137.329,A -85,B 0,C 180,E1 -4320,E2 -4320} C_VEL
LIN {X 0,Y 531.127,Z 137.325,A -85,B 0,C 180,E1 -4322.275,E2 -4322.275} C_VEL
LIN {X 0,Y 531.075,Z 137.328,A -85,B 0,C 180,E1 -4325.316,E2 -4325.316} C_VEL
LIN {X 0,Y 530.976,Z 137.342,A -85,B 0,C 180,E1 -4328.372,E2 -4328.372} C_VEL
LIN {X 0,Y 531.005,Z 137.342,A -85,B 0,C 180,E1 -4331.65,E2 -4331.65} C_VEL
LIN {X 0,Y 531.013,Z 137.335,A -85,B 0,C 180,E1 -4334.951,E2 -4334.951} C_VEL
LIN {X 0,Y 530.965,Z 137.349,A -85,B 0,C 180,E1 -4337.724,E2 -4337.724} C_VEL
LIN {X 0,Y 530.965,Z 137.343,A -85,B 0,C 180,E1 -4340.13,E2 -4340.13} C_VEL
LIN {X 0,Y 530.911,Z 137.347,A -85,B 0,C 180,E1 -4342.575,E2 -4342.575} C_VEL
LIN {X 0,Y 530.942,Z 137.346,A -85,B 0,C 180,E1 -4345.061,E2 -4345.061} C_VEL
LIN {X 0,Y 530.945,Z 137.35,A -85,B 0,C 180,E1 -4347.6,E2 -4347.6} C_VEL
LIN {X 0,Y 530.937,Z 137.345,A -85,B 0,C 180,E1 -4350.639,E2 -4350.639} C_VEL
LIN {X 0,Y 530.957,Z 137.348,A -85,B 0,C 180,E1 -4353.5,E2 -4353.5} C_VEL
LIN {X 0,Y 530.904,Z 137.348,A -85,B 0,C 180,E1 -4356.148,E2 -4356.148} C_VEL
LIN {X 0,Y 530.952,Z 137.344,A -85,B 0,C 180,E1 -4358.652,E2 -4358.652} C_VEL
LIN {X 0,Y 530.945,Z 137.348,A -85,B 0,C 180,E1 -4361.441,E2 -4361.441} C_VEL
LIN {X 0,Y 530.96,Z 137.343,A -85,B 0,C 180,E1 -4364.55,E2 -4364.55} C_VEL
LIN {X 0,Y 530.911,Z 137.349,A -85,B 0,C 180,E1 -4367.537,E2 -4367.537} C_VEL
LIN {X 0,Y 530.951,Z 137.346,A -85,B 0,C 180,E1 -4370.554,E2 -4370.554} C_VEL
LIN {X 0,Y 530.905,Z 137.35,A -85,B 0,C 180,E1 -4373.438,E2 -4373.438} C_VEL
LIN {X 0,Y 530.948,Z 137.344,A -85,B 0,C 180,E1 -4376.225,E2 -4376.225} C_VEL
LIN {X 0,Y 530.934,Z 137.351,A -85,B 0,C 180,E1 -4378.92,E2 -4378.92} C_VEL
LIN {X 0,Y 530.929,Z 137.346,A -85,B 0,C 180,E1 -4381.541,E2 -4381.541} C_VEL
LIN {X 0,Y 530.927,Z 137.348,A -85,B 0,C 180,E1 -4384.176,E2 -4384.176} C_VEL
LIN {X 0,Y 530.955,Z 137.538,A -85,B 0,C 180,E1 -4386.059,E2 -4386.059} C_VEL
LIN {X 0,Y 532.218,Z 144.71,A -85,B 0,C 180,E1 -4387.279,E2 -4387.279} C_VEL
LIN {X 0,Y 531.948,Z 160.038,A -85,B 0,C 180,E1 -4389.726,E2 -4389.726} C_VEL
LIN {X 0,Y 531.58,Z 176.437,A -85,B 0,C 180,E1 -4392.297,E2 -4392.297} C_VEL
LIN {X 0,Y 531.27,Z 194.155,A -85,B 0,C 180,E1 -4395.051,E2 -4395.051} C_VEL
LIN {X 0,Y 532.761,Z 205.404,A -85,B 0,C 180,E1 -4395.253,E2 -4395.253} C_VEL
LIN {X 0,Y 532.353,Z 302.463,A -85,B 0,C 180,E1 -4396.594,E2 -4396.594} C_VEL
LIN {X 0,Y 532.184,Z 315.655,A -85,B 0,C 180,E1 -4396.929,E2 -4396.929} C_VEL
LIN {X 0,Y 531.935,Z 328.347,A -85,B 0,C 180,E1 -4397.408,E2 -4397.408} C_VEL
LIN {X 0,Y 531.664,Z 340.149,A -85,B 0,C 180,E1 -4398.015,E2 -4398.015} C_VEL
LIN {X 0,Y 531.477,Z 351.307,A -85,B 0,C 180,E1 -4398.753,E2 -4398.753} C_VEL
LIN {X 0,Y 531.21,Z 361.806,A -85,B 0,C 180,E1 -4399.615,E2 -4399.615} C_VEL
LIN {X 0,Y 531.015,Z 370.387,A -85,B 0,C 180,E1 -4400.477,E2 -4400.477} C_VEL
LIN {X 0,Y 530.849,Z 378.302,A -85,B 0,C 180,E1 -4401.434,E2 -4401.434} C_VEL
LIN {X 0,Y 530.668,Z 386.029,A -85,B 0,C 180,E1 -4402.581,E2 -4402.581} C_VEL
LIN {X 0,Y 530.575,Z 393.144,A -85,B 0,C 180,E1 -4403.917,E2 -4403.917} C_VEL
LIN {X 0,Y 530.459,Z 397.875,A -85,B 0,C 180,E1 -4405.06,E2 -4405.06} C_VEL
LIN {X 0,Y 530.516,Z 401.493,A -85,B 0,C 180,E1 -4406.202,E2 -4406.202} C_VEL
LIN {X 0,Y 530.457,Z 403.357,A -85,B 0,C 180,E1 -4406.962,E2 -4406.962} C_VEL
LIN {X 0,Y 530.411,Z 404.753,A -85,B 0,C 180,E1 -4407.722,E2 -4407.722} C_VEL
LIN {X 0,Y 530.347,Z 406.356,A -85,B 0,C 180,E1 -4409.241,E2 -4409.241} C_VEL
LIN {X 0,Y 530.348,Z 406.572,A -85,B 0,C 180,E1 -4410,E2 -4410} C_VEL
LIN {X 0,Y 530.361,Z 405.745,A -85,B 0,C 180,E1 -4411.519,E2 -4411.519} C_VEL
LIN {X 0,Y 530.411,Z 404.749,A -85,B 0,C 180,E1 -4412.278,E2 -4412.278} C_VEL
LIN {X 0,Y 530.457,Z 403.348,A -85,B 0,C 180,E1 -4413.038,E2 -4413.038} C_VEL
LIN {X 0,Y 530.521,Z 400.406,A -85,B 0,C 180,E1 -4414.178,E2 -4414.178} C_VEL
LIN {X 0,Y 530.522,Z 396.419,A -85,B 0,C 180,E1 -4415.321,E2 -4415.321} C_VEL
LIN {X 0,Y 530.582,Z 390.763,A -85,B 0,C 180,E1 -4416.566,E2 -4416.566} C_VEL
LIN {X 0,Y 530.705,Z 383.584,A -85,B 0,C 180,E1 -4417.801,E2 -4417.801} C_VEL
LIN {X 0,Y 530.887,Z 375.262,A -85,B 0,C 180,E1 -4418.948,E2 -4418.948} C_VEL
LIN {X 0,Y 531.063,Z 366.721,A -85,B 0,C 180,E1 -4419.906,E2 -4419.906} C_VEL
LIN {X 0,Y 531.342,Z 356.17,A -85,B 0,C 180,E1 -4420.864,E2 -4420.864} C_VEL
LIN {X 0,Y 531.607,Z 344.315,A -85,B 0,C 180,E1 -4421.725,E2 -4421.725} C_VEL
LIN {X 0,Y 531.867,Z 332.279,A -85,B 0,C 180,E1 -4422.399,E2 -4422.399} C_VEL
LIN {X 0,Y 532.068,Z 319.781,A -85,B 0,C 180,E1 -4422.928,E2 -4422.928} C_VEL
LIN {X 0,Y 532.286,Z 306.801,A -85,B 0,C 180,E1 -4423.311,E2 -4423.311} C_VEL
LIN {X 0,Y 532.457,Z 291.205,A -85,B 0,C 180,E1 -4423.573,E2 -4423.573} C_VEL
LIN {X 0,Y 532.636,Z 203.192,A -85,B 0,C 180,E1 -4424.78,E2 -4424.78} C_VEL
LIN {X 0,Y 531.239,Z 193.84,A -85,B 0,C 180,E1 -4424.965,E2 -4424.965} C_VEL
LIN {X 0,Y 531.56,Z 175.191,A -85,B 0,C 180,E1 -4427.834,E2 -4427.834} C_VEL
LIN {X 0,Y 531.986,Z 155.507,A -85,B 0,C 180,E1 -4430.897,E2 -4430.897} C_VEL
LIN {X 0,Y 532.114,Z 143.922,A -85,B 0,C 180,E1 -4432.726,E2 -4432.726} C_VEL
LIN {X 0,Y 530.948,Z 137.35,A -85,B 0,C 180,E1 -4433.85,E2 -4433.85} C_VEL
LIN {X 0,Y 530.94,Z 137.348,A -85,B 0,C 180,E1 -4436.747,E2 -4436.747} C_VEL
LIN {X 0,Y 530.914,Z 137.359,A -85,B 0,C 180,E1 -4439.326,E2 -4439.326} C_VEL
LIN {X 0,Y 530.95,Z 137.345,A -85,B 0,C 180,E1 -4442.097,E2 -4442.097} C_VEL
LIN {X 0,Y 530.952,Z 137.348,A -85,B 0,C 180,E1 -4444.848,E2 -4444.848} C_VEL
LIN {X 0,Y 530.927,Z 137.351,A -85,B 0,C 180,E1 -4447.51,E2 -4447.51} C_VEL
LIN {X 0,Y 530.932,Z 137.348,A -85,B 0,C 180,E1 -4450.437,E2 -4450.437} C_VEL
LIN {X 0,Y 530.922,Z 137.35,A -85,B 0,C 180,E1 -4453.498,E2 -4453.498} C_VEL
LIN {X 0,Y 530.96,Z 137.343,A -85,B 0,C 180,E1 -4455.623,E2 -4455.623} C_VEL
LIN {X 0,Y 530.923,Z 137.353,A -85,B 0,C 180,E1 -4458.983,E2 -4458.983} C_VEL
LIN {X 0,Y 530.94,Z 137.345,A -85,B 0,C 180,E1 -4461.528,E2 -4461.528} C_VEL
LIN {X 0,Y 530.924,Z 137.349,A -85,B 0,C 180,E1 -4464.377,E2 -4464.377} C_VEL
LIN {X 0,Y 530.958,Z 137.344,A -85,B 0,C 180,E1 -4467.132,E2 -4467.132} C_VEL
LIN {X 0,Y 530.922,Z 137.345,A -85,B 0,C 180,E1 -4469.8,E2 -4469.8} C_VEL
LIN {X 0,Y 530.947,Z 137.351,A -85,B 0,C 180,E1 -4472.479,E2 -4472.479} C_VEL
LIN {X 0,Y 530.94,Z 137.347,A -85,B 0,C 180,E1 -4474.939,E2 -4474.939} C_VEL
LIN {X 0,Y 530.94,Z 137.348,A -85,B 0,C 180,E1 -4478.245,E2 -4478.245} C_VEL
LIN {X 0,Y 530.932,Z 137.348,A -85,B 0,C 180,E1 -4480.675,E2 -4480.675} C_VEL
LIN {X 0,Y 530.928,Z 137.346,A -85,B 0,C 180,E1 -4483.069,E2 -4483.069} C_VEL
LIN {X 0,Y 530.99,Z 137.337,A -85,B 0,C 180,E1 -4485.435,E2 -4485.435} C_VEL
LIN {X 0,Y 530.977,Z 137.343,A -85,B 0,C 180,E1 -4488.548,E2 -4488.548} C_VEL
LIN {X 0,Y 530.974,Z 137.342,A -85,B 0,C 180,E1 -4491.628,E2 -4491.628} C_VEL
LIN {X 0,Y 531.073,Z 137.327,A -85,B 0,C 180,E1 -4494.684,E2 -4494.684} C_VEL
LIN {X 0,Y 531.125,Z 137.326,A -85,B 0,C 180,E1 -4497.725,E2 -4497.725} C_VEL
LIN {X 0,Y 531.119,Z 137.329,A -85,B 0,C 180,E1 -4500,E2 -4500} C_VEL
LIN {X 0,Y 531.125,Z 137.325,A -85,B 0,C 180,E1 -4502.275,E2 -4502.275} C_VEL
LIN {X 0,Y 531.073,Z 137.33,A -85,B 0,C 180,E1 -4505.315,E2 -4505.315} C_VEL
LIN {X 0,Y 530.973,Z 137.343,A -85,B 0,C 180,E1 -4508.372,E2 -4508.372} C_VEL
LIN {X 0,Y 531.002,Z 137.346,A -85,B 0,C 180,E1 -4511.65,E2 -4511.65} C_VEL
LIN {X 0,Y 531.011,Z 137.339,A -85,B 0,C 180,E1 -4514.951,E2 -4514.951} C_VEL
LIN {X 0,Y 530.953,Z 137.344,A -85,B 0,C 180,E1 -4518.522,E2 -4518.522} C_VEL
LIN {X 0,Y 530.961,Z 137.346,A -85,B 0,C 180,E1 -4520.939,E2 -4520.939} C_VEL
LIN {X 0,Y 531.005,Z 137.413,A -85,B 0,C 180,E1 -4523.81,E2 -4523.81} C_VEL
LIN {X 0,Y 531.528,Z 141.782,A -85,B 0,C 180,E1 -4524.614,E2 -4524.614} C_VEL
LIN {X 0,Y 531.354,Z 156.029,A -85,B 0,C 180,E1 -4527.149,E2 -4527.149} C_VEL
LIN {X 0,Y 531.264,Z 166.866,A -85,B 0,C 180,E1 -4529.096,E2 -4529.096} C_VEL
LIN {X 0,Y 532.849,Z 176.455,A -85,B 0,C 180,E1 -4529.291,E2 -4529.291} C_VEL
LIN {X 0,Y 532.365,Z 274.751,A -85,B 0,C 180,E1 -4530.657,E2 -4530.657} C_VEL
LIN {X 0,Y 532.311,Z 280.227,A -85,B 0,C 180,E1 -4530.779,E2 -4530.779} C_VEL
LIN {X 0,Y 531.438,Z 285.939,A -85,B 0,C 180,E1 -4530.92,E2 -4530.92} C_VEL
LIN {X 0,Y 528.406,Z 295.121,A -85,B 0,C 180,E1 -4531.168,E2 -4531.168} C_VEL
LIN {X 0,Y 525.576,Z 304.113,A -85,B 0,C 180,E1 -4531.504,E2 -4531.504} C_VEL
LIN {X 0,Y 524.906,Z 309.383,A -85,B 0,C 180,E1 -4531.77,E2 -4531.77} C_VEL
LIN {X 0,Y 524.585,Z 320.806,A -85,B 0,C 180,E1 -4532.496,E2 -4532.496} C_VEL
LIN {X 0,Y 524.308,Z 331.24,A -85,B 0,C 180,E1 -4533.338,E2 -4533.338} C_VEL
LIN {X 0,Y 524.098,Z 340.712,A -85,B 0,C 180,E1 -4534.278,E2 -4534.278} C_VEL
LIN {X 0,Y 523.875,Z 348.638,A -85,B 0,C 180,E1 -4535.23,E2 -4535.23} C_VEL
LIN {X 0,Y 523.714,Z 356.45,A -85,B 0,C 180,E1 -4536.374,E2 -4536.374} C_VEL
LIN {X 0,Y 523.54,Z 363.221,A -85,B 0,C 180,E1 -4537.627,E2 -4537.627} C_VEL
LIN {X 0,Y 523.454,Z 368.415,A -85,B 0,C 180,E1 -4538.858,E2 -4538.858} C_VEL
LIN {X 0,Y 523.389,Z 372.469,A -85,B 0,C 180,E1 -4540.131,E2 -4540.131} C_VEL
LIN {X 0,Y 523.333,Z 375.007,A -85,B 0,C 180,E1 -4541.234,E2 -4541.234} C_VEL
LIN {X 0,Y 523.283,Z 376.738,A -85,B 0,C 180,E1 -4542.382,E2 -4542.382} C_VEL
LIN {X 0,Y 523.27,Z 377.564,A -85,B 0,C 180,E1 -4543.51,E2 -4543.51} C_VEL
LIN {X 0,Y 523.308,Z 377.543,A -85,B 0,C 180,E1 -4544.621,E2 -4544.621} C_VEL
LIN {X 0,Y 523.304,Z 376.726,A -85,B 0,C 180,E1 -4545.705,E2 -4545.705} C_VEL
LIN {X 0,Y 523.308,Z 375.148,A -85,B 0,C 180,E1 -4546.771,E2 -4546.771} C_VEL
LIN {X 0,Y 523.37,Z 372.812,A -85,B 0,C 180,E1 -4547.824,E2 -4547.824} C_VEL
LIN {X 0,Y 523.431,Z 369.72,A -85,B 0,C 180,E1 -4548.86,E2 -4548.86} C_VEL
LIN {X 0,Y 523.512,Z 364.521,A -85,B 0,C 180,E1 -4550.172,E2 -4550.172} C_VEL
LIN {X 0,Y 523.653,Z 358.75,A -85,B 0,C 180,E1 -4551.312,E2 -4551.312} C_VEL
LIN {X 0,Y 523.829,Z 350.513,A -85,B 0,C 180,E1 -4552.604,E2 -4552.604} C_VEL
LIN {X 0,Y 524.044,Z 341.598,A -85,B 0,C 180,E1 -4553.71,E2 -4553.71} C_VEL
LIN {X 0,Y 524.322,Z 331.884,A -85,B 0,C 180,E1 -4554.688,E2 -4554.688} C_VEL
LIN {X 0,Y 524.589,Z 321.627,A -85,B 0,C 180,E1 -4555.527,E2 -4555.527} C_VEL
LIN {X 0,Y 524.864,Z 309.527,A -85,B 0,C 180,E1 -4556.31,E2 -4556.31} C_VEL
LIN {X 0,Y 525.139,Z 297.158,A -85,B 0,C 180,E1 -4556.918,E2 -4556.918} C_VEL
LIN {X 0,Y 525.316,Z 284.368,A -85,B 0,C 180,E1 -4557.375,E2 -4557.375} C_VEL
LIN {X 0,Y 525.5,Z 271.293,A -85,B 0,C 180,E1 -4557.674,E2 -4557.674} C_VEL
LIN {X 0,Y 525.873,Z 175.935,A -85,B 0,C 180,E1 -4559.012,E2 -4559.012} C_VEL
LIN {X 0,Y 524.287,Z 167.074,A -85,B 0,C 180,E1 -4559.19,E2 -4559.19} C_VEL
LIN {X 0,Y 524.552,Z 151.175,A -85,B 0,C 180,E1 -4562.161,E2 -4562.161} C_VEL
LIN {X 0,Y 524.659,Z 142.386,A -85,B 0,C 180,E1 -4563.829,E2 -4563.829} C_VEL
LIN {X 0,Y 523.934,Z 138.225,A -85,B 0,C 180,E1 -4564.687,E2 -4564.687} C_VEL
LIN {X 0,Y 523.915,Z 138.222,A -85,B 0,C 180,E1 -4567.939,E2 -4567.939} C_VEL
LIN {X 0,Y 523.947,Z 138.223,A -85,B 0,C 180,E1 -4570.407,E2 -4570.407} C_VEL
LIN {X 0,Y 523.914,Z 138.223,A -85,B 0,C 180,E1 -4572.836,E2 -4572.836} C_VEL
LIN {X 0,Y 523.959,Z 138.214,A -85,B 0,C 180,E1 -4575.236,E2 -4575.236} C_VEL
LIN {X 0,Y 523.955,Z 138.222,A -85,B 0,C 180,E1 -4578.393,E2 -4578.393} C_VEL
LIN {X 0,Y 523.942,Z 138.216,A -85,B 0,C 180,E1 -4581.515,E2 -4581.515} C_VEL
LIN {X 0,Y 524.025,Z 138.208,A -85,B 0,C 180,E1 -4584.613,E2 -4584.613} C_VEL
LIN {X 0,Y 524.1,Z 138.199,A -85,B 0,C 180,E1 -4587.695,E2 -4587.695} C_VEL
LIN {X 0,Y 524.093,Z 138.204,A -85,B 0,C 180,E1 -4590,E2 -4590} C_VEL
LIN {X 0,Y 524.1,Z 138.201,A -85,B 0,C 180,E1 -4592.306,E2 -4592.306} C_VEL
LIN {X 0,Y 523.997,Z 138.214,A -85,B 0,C 180,E1 -4596.16,E2 -4596.16} C_VEL
LIN {X 0,Y 523.94,Z 138.217,A -85,B 0,C 180,E1 -4599.263,E2 -4599.263} C_VEL
LIN {X 0,Y 523.94,Z 138.217,A -85,B 0,C 180,E1 -4602.393,E2 -4602.393} C_VEL
LIN {X 0,Y 523.908,Z 138.226,A -85,B 0,C 180,E1 -4605.563,E2 -4605.563} C_VEL
LIN {X 0,Y 523.909,Z 138.22,A -85,B 0,C 180,E1 -4608.781,E2 -4608.781} C_VEL
LIN {X 0,Y 523.899,Z 138.224,A -85,B 0,C 180,E1 -4611.235,E2 -4611.235} C_VEL
LIN {X 0,Y 523.927,Z 138.218,A -85,B 0,C 180,E1 -4614.196,E2 -4614.196} C_VEL
LIN {X 0,Y 523.888,Z 138.226,A -85,B 0,C 180,E1 -4617.136,E2 -4617.136} C_VEL
LIN {X 0,Y 523.861,Z 138.23,A -85,B 0,C 180,E1 -4619.761,E2 -4619.761} C_VEL
LIN {X 0,Y 523.925,Z 138.218,A -85,B 0,C 180,E1 -4622.45,E2 -4622.45} C_VEL
LIN {X 0,Y 523.903,Z 138.228,A -85,B 0,C 180,E1 -4625.228,E2 -4625.228} C_VEL
LIN {X 0,Y 523.904,Z 138.22,A -85,B 0,C 180,E1 -4628.102,E2 -4628.102} C_VEL
LIN {X 0,Y 523.905,Z 138.227,A -85,B 0,C 180,E1 -4631.304,E2 -4631.304} C_VEL
LIN {X 0,Y 523.927,Z 138.221,A -85,B 0,C 180,E1 -4634.689,E2 -4634.689} C_VEL
LIN {X 0,Y 523.888,Z 138.222,A -85,B 0,C 180,E1 -4637.875,E2 -4637.875} C_VEL
LIN {X 0,Y 523.903,Z 138.229,A -85,B 0,C 180,E1 -4640.914,E2 -4640.914} C_VEL
LIN {X 0,Y 523.856,Z 138.226,A -85,B 0,C 180,E1 -4643.822,E2 -4643.822} C_VEL
LIN {X 0,Y 523.905,Z 138.226,A -85,B 0,C 180,E1 -4646.633,E2 -4646.633} C_VEL
LIN {X 0,Y 523.904,Z 138.222,A -85,B 0,C 180,E1 -4649.353,E2 -4649.353} C_VEL
LIN {X 0,Y 523.904,Z 138.224,A -85,B 0,C 180,E1 -4652.295,E2 -4652.295} C_VEL
LIN {X 0,Y 523.893,Z 138.222,A -85,B 0,C 180,E1 -4655.427,E2 -4655.427} C_VEL
LIN {X 0,Y 523.915,Z 138.224,A -85,B 0,C 180,E1 -4658.766,E2 -4658.766} C_VEL
LIN {X 0,Y 523.917,Z 138.219,A -85,B 0,C 180,E1 -4661.22,E2 -4661.22} C_VEL
LIN {X 0,Y 523.872,Z 138.224,A -85,B 0,C 180,E1 -4663.637,E2 -4663.637} C_VEL
LIN {X 0,Y 523.956,Z 138.214,A -85,B 0,C 180,E1 -4665.235,E2 -4665.235} C_VEL
LIN {X 0,Y 523.952,Z 138.222,A -85,B 0,C 180,E1 -4668.393,E2 -4668.393} C_VEL
LIN {X 0,Y 523.938,Z 138.216,A -85,B 0,C 180,E1 -4671.515,E2 -4671.515} C_VEL
LIN {X 0,Y 524.022,Z 138.208,A -85,B 0,C 180,E1 -4674.613,E2 -4674.613} C_VEL
LIN {X 0,Y 524.097,Z 138.199,A -85,B 0,C 180,E1 -4677.695,E2 -4677.695} C_VEL
LIN {X 0,Y 524.09,Z 138.205,A -85,B 0,C 180,E1 -4680,E2 -4680} C_VEL
LIN {X 0,Y 524.097,Z 138.201,A -85,B 0,C 180,E1 -4682.306,E2 -4682.306} C_VEL
LIN {X 0,Y 523.994,Z 138.214,A -85,B 0,C 180,E1 -4686.16,E2 -4686.16} C_VEL
LIN {X 0,Y 523.938,Z 138.217,A -85,B 0,C 180,E1 -4689.263,E2 -4689.263} C_VEL
LIN {X 0,Y 523.937,Z 138.217,A -85,B 0,C 180,E1 -4692.394,E2 -4692.394} C_VEL
LIN {X 0,Y 523.906,Z 138.227,A -85,B 0,C 180,E1 -4695.563,E2 -4695.563} C_VEL
LIN {X 0,Y 523.907,Z 138.22,A -85,B 0,C 180,E1 -4698.781,E2 -4698.781} C_VEL
LIN {X 0,Y 523.897,Z 138.225,A -85,B 0,C 180,E1 -4701.236,E2 -4701.236} C_VEL
LIN {X 0,Y 523.927,Z 138.218,A -85,B 0,C 180,E1 -4704.196,E2 -4704.196} C_VEL
LIN {X 0,Y 523.888,Z 138.227,A -85,B 0,C 180,E1 -4707.137,E2 -4707.137} C_VEL
LIN {X 0,Y 523.861,Z 138.229,A -85,B 0,C 180,E1 -4709.761,E2 -4709.761} C_VEL
LIN {X 0,Y 523.925,Z 138.218,A -85,B 0,C 180,E1 -4712.45,E2 -4712.45} C_VEL
LIN {X 0,Y 523.903,Z 138.229,A -85,B 0,C 180,E1 -4715.228,E2 -4715.228} C_VEL
LIN {X 0,Y 523.896,Z 138.221,A -85,B 0,C 180,E1 -4718.104,E2 -4718.104} C_VEL
LIN {X 0,Y 523.882,Z 138.232,A -85,B 0,C 180,E1 -4721.098,E2 -4721.098} C_VEL
LIN {X 0,Y 523.916,Z 138.219,A -85,B 0,C 180,E1 -4724.231,E2 -4724.231} C_VEL
LIN {X 0,Y 523.877,Z 138.23,A -85,B 0,C 180,E1 -4726.829,E2 -4726.829} C_VEL
LIN {X 0,Y 523.911,Z 138.219,A -85,B 0,C 180,E1 -4729.918,E2 -4729.918} C_VEL
LIN {X 0,Y 523.868,Z 138.234,A -85,B 0,C 180,E1 -4732.865,E2 -4732.865} C_VEL
LIN {X 0,Y 523.909,Z 138.22,A -85,B 0,C 180,E1 -4735.708,E2 -4735.708} C_VEL
LIN {X 0,Y 523.904,Z 138.225,A -85,B 0,C 180,E1 -4738.455,E2 -4738.455} C_VEL
LIN {X 0,Y 523.871,Z 138.228,A -85,B 0,C 180,E1 -4741.122,E2 -4741.122} C_VEL
LIN {X 0,Y 523.88,Z 138.225,A -85,B 0,C 180,E1 -4744.004,E2 -4744.004} C_VEL
LIN {X 0,Y 523.925,Z 138.341,A -85,B 0,C 180,E1 -4745.878,E2 -4745.878} C_VEL
LIN {X 0,Y 525.254,Z 145.818,A -85,B 0,C 180,E1 -4747.169,E2 -4747.169} C_VEL
LIN {X 0,Y 524.972,Z 161.028,A -85,B 0,C 180,E1 -4749.631,E2 -4749.631} C_VEL
LIN {X 0,Y 524.603,Z 176.253,A -85,B 0,C 180,E1 -4752.054,E2 -4752.054} C_VEL
LIN {X 0,Y 524.25,Z 193.968,A -85,B 0,C 180,E1 -4754.845,E2 -4754.845} C_VEL
LIN {X 0,Y 525.875,Z 204.834,A -85,B 0,C 180,E1 -4755.05,E2 -4755.05} C_VEL
LIN {X 0,Y 525.447,Z 302.056,A -85,B 0,C 180,E1 -4756.414,E2 -4756.414} C_VEL
LIN {X 0,Y 525.254,Z 315.313,A -85,B 0,C 180,E1 -4756.754,E2 -4756.754} C_VEL
LIN {X 0,Y 525.007,Z 328.044,A -85,B 0,C 180,E1 -4757.24,E2 -4757.24} C_VEL
LIN {X 0,Y 524.698,Z 340.086,A -85,B 0,C 180,E1 -4757.866,E2 -4757.866} C_VEL
LIN {X 0,Y 524.485,Z 351.053,A -85,B 0,C 180,E1 -4758.601,E2 -4758.601} C_VEL
LIN {X 0,Y 524.206,Z 361.564,A -85,B 0,C 180,E1 -4759.475,E2 -4759.475} C_VEL
LIN {X 0,Y 523.96,Z 370.155,A -85,B 0,C 180,E1 -4760.348,E2 -4760.348} C_VEL
LIN {X 0,Y 523.779,Z 378.079,A -85,B 0,C 180,E1 -4761.318,E2 -4761.318} C_VEL
LIN {X 0,Y 523.596,Z 385.816,A -85,B 0,C 180,E1 -4762.48,E2 -4762.48} C_VEL
LIN {X 0,Y 523.47,Z 392.936,A -85,B 0,C 180,E1 -4763.834,E2 -4763.834} C_VEL
LIN {X 0,Y 523.383,Z 397.674,A -85,B 0,C 180,E1 -4764.993,E2 -4764.993} C_VEL
LIN {X 0,Y 523.443,Z 401.295,A -85,B 0,C 180,E1 -4766.151,E2 -4766.151} C_VEL
LIN {X 0,Y 523.368,Z 403.16,A -85,B 0,C 180,E1 -4766.921,E2 -4766.921} C_VEL
LIN {X 0,Y 523.335,Z 404.559,A -85,B 0,C 180,E1 -4767.691,E2 -4767.691} C_VEL
LIN {X 0,Y 523.253,Z 406.162,A -85,B 0,C 180,E1 -4769.23,E2 -4769.23} C_VEL
LIN {X 0,Y 523.251,Z 406.377,A -85,B 0,C 180,E1 -4770,E2 -4770} C_VEL
LIN {X 0,Y 523.275,Z 405.549,A -85,B 0,C 180,E1 -4771.539,E2 -4771.539} C_VEL
LIN {X 0,Y 523.335,Z 404.55,A -85,B 0,C 180,E1 -4772.309,E2 -4772.309} C_VEL
LIN {X 0,Y 523.367,Z 403.147,A -85,B 0,C 180,E1 -4773.079,E2 -4773.079} C_VEL
LIN {X 0,Y 523.422,Z 400.199,A -85,B 0,C 180,E1 -4774.235,E2 -4774.235} C_VEL
LIN {X 0,Y 523.456,Z 396.207,A -85,B 0,C 180,E1 -4775.393,E2 -4775.393} C_VEL
LIN {X 0,Y 523.501,Z 391.034,A -85,B 0,C 180,E1 -4776.559,E2 -4776.559} C_VEL
LIN {X 0,Y 523.628,Z 384.592,A -85,B 0,C 180,E1 -4777.713,E2 -4777.713} C_VEL
LIN {X 0,Y 523.793,Z 376.519,A -85,B 0,C 180,E1 -4778.876,E2 -4778.876} C_VEL
LIN {X 0,Y 524.003,Z 368.284,A -85,B 0,C 180,E1 -4779.846,E2 -4779.846} C_VEL
LIN {X 0,Y 524.303,Z 358.238,A -85,B 0,C 180,E1 -4780.816,E2 -4780.816} C_VEL
LIN {X 0,Y 524.586,Z 346.958,A -85,B 0,C 180,E1 -4781.684,E2 -4781.684} C_VEL
